// ---- 20_Product/10_BCF/10_Base/11_Com/01_Stringhandling/F_StringToTimeDate.TcPOU
// HI = parsing string 'Y-M-D, h:m:s.ms' or 'Y-M-D Th:m:s.ms' to TIMESTRUCT successful
FUNCTION PUBLIC F_StringToTimeDate : BOOL
(**************************************************************************************
 * 	Application		:	BoxControl Framework
 *	Revision		  :	$Revision: 461868 $
 *	Revision date	:	$Date: 1979-01-09 14:35:13 +0200 (Di., 09 Jan 1979) $
 *	Last changed by	:	$Author: b7lipim $
 *	URL				:	$URL: http://almscdc.swisslog.com/repo/SWPD/Development/BoxControlFramework/20_Release/branches/R1.x/01_Software/BCF/BCF/JumpStart/20_Product/10_BCF/10_Base/11_Com/12_DebugMsg/00_GVLs/DebugTextBlocks.TcGVL $
 *
 * ------------------------------------------------------------------------------------
 *	Copyright Swisslog [IP AG], Switzerland. All rights reserved.
 * 
 * ------------------------------------------------------------------------------------
 *	
 * 	Revision History: 
 *
 *  VERSION DATE         INITIALS     DESCRIPTION
 *  0.0     DD.MM.YYYY   (name)       (explain customized modifications)
 *
 **************************************************************************************)

(********************************************************************************************************************************)
VAR_INPUT
  DestStart             : POINTER TO BYTE                  := 0;     // = ADR(MyString)                    -> start position to concat
  DestEnd               : POINTER TO BYTE                  := 0;     // = ADR(MyString) + SIZEOF(MyString) -> buffer/string end
  (*----------------------------------------------------------------------------------------------------------------------------*)
  AllowInvalidChars     : BOOL                             := FALSE; // HI = ignore invalid char
END_VAR

(********************************************************************************************************************************)
VAR_OUTPUT
  Result                : TIMESTRUCT;                                     // parsing result
END_VAR

(********************************************************************************************************************************)
VAR
  Char                  : BYTE                             := 0;
  ItemType              : BYTE                             := UNDEF;
END_VAR

(********************************************************************************************************************************)
VAR CONSTANT
  UNDEF                 : BYTE := 0;
  YEAR                  : BYTE := 1;
  MONTH                 : BYTE := 2;
  DAY                   : BYTE := 3;
  HOUR                  : BYTE := 4;
  MINUTE                : BYTE := 5;
  SECOND                : BYTE := 6;
  MSEC                  : BYTE := 7;
END_VAR


(********************************************************************************************************************************)
(** check inputs ****************************************************************************************************************)
IF (    ( DestStart = 0 )
     OR ( DestEnd   = 0 )  )
THEN
  F_StringToTimeDate:= FALSE;
  RETURN;
END_IF




(********************************************************************************************************************************)
(********************************************************************************************************************************)
ItemType    := YEAR;

WHILE(DestStart^ <> 16#00)
DO
  Char     := DestStart^;
  DestStart:= DestStart + SIZEOF(DestStart^);
  (*-- numbers ----------------------------------------------------------------------------------------------*)
  IF (     ( Char >= 16#30 )
       AND ( Char <= 16#39 )  )
  THEN
    IF   (ItemType          = YEAR  ) THEN  Result.wYear        := (Result.wYear         * WORD#10) + BYTE_TO_WORD(Char - 16#30); 
    ELSIF(ItemType          = MONTH ) THEN  Result.wMonth       := (Result.wMonth        * WORD#10) + BYTE_TO_WORD(Char - 16#30);
    ELSIF(ItemType          = DAY   ) THEN  Result.wDay         := (Result.wDay          * WORD#10) + BYTE_TO_WORD(Char - 16#30);
    ELSIF(ItemType          = HOUR  ) THEN  Result.wHour        := (Result.wHour         * WORD#10) + BYTE_TO_WORD(Char - 16#30);
    ELSIF(ItemType          = MINUTE) THEN  Result.wMinute      := (Result.wMinute       * WORD#10) + BYTE_TO_WORD(Char - 16#30);
    ELSIF(ItemType          = SECOND) THEN  Result.wSecond      := (Result.wSecond       * WORD#10) + BYTE_TO_WORD(Char - 16#30);
    ELSIF(ItemType          = MSEC  ) THEN  Result.wMilliseconds:= (Result.wMilliseconds * WORD#10) + BYTE_TO_WORD(Char - 16#30);
    ELSIF(AllowInvalidChars = FALSE ) THEN  F_StringToTimeDate:= FALSE;  RETURN;
    END_IF

  (*-- separation during date -------------------------------------------------------------------------------*)
  ELSIF( Char = 16#2D ) (* '-' *)
  THEN
    IF   (ItemType          = YEAR  ) THEN  ItemType:= MONTH; 
    ELSIF(ItemType          = MONTH ) THEN  ItemType:= DAY;
    ELSIF(AllowInvalidChars = FALSE ) THEN  F_StringToTimeDate:= FALSE;  RETURN;
    END_IF

  (*-- separation date->time --------------------------------------------------------------------------------*)
  ELSIF(    ( Char = 16#2C )    (* ',' *)
         OR ( Char = 16#54 )  ) (* 'T' *)
  THEN
    IF   (ItemType          = DAY   ) THEN  ItemType:= HOUR; 
    ELSIF(AllowInvalidChars = FALSE ) THEN  F_StringToTimeDate:= FALSE;  RETURN;
    END_IF

  (*-- separation during time -------------------------------------------------------------------------------*)
  ELSIF( Char = 16#3A ) (* ':' *)
  THEN
    IF   (ItemType          = HOUR   ) THEN  ItemType:= MINUTE; 
    ELSIF(ItemType          = MINUTE ) THEN  ItemType:= SECOND;
    ELSIF(AllowInvalidChars = FALSE  ) THEN  F_StringToTimeDate:= FALSE;  RETURN;
    END_IF

  (*-- separation during time -------------------------------------------------------------------------------*)
  ELSIF( Char = 16#2E ) (* '.' *)
  THEN
    IF   (ItemType          = SECOND ) THEN  ItemType:= MSEC; 
    ELSIF(AllowInvalidChars = FALSE  ) THEN  F_StringToTimeDate:= FALSE;  RETURN;
    END_IF

  (*-- always ignore spaces ---------------------------------------------------------------------------------*)
  ELSIF( Char = 16#20) (* ' ' *)
  THEN
    CONTINUE;

  (*---------------------------------------------------------------------------------------------------------*)
  ELSIF (AllowInvalidChars = FALSE )
  THEN
    F_StringToTimeDate:= FALSE;
    RETURN;
  END_IF

END_WHILE




(********************************************************************************************************************************)
(** done ************************************************************************************************************************)
F_StringToTimeDate:=TRUE;

END_FUNCTION

// ---- 20_Product/30_Toolbox/12_StringStream/F_AssembleByteStream.TcPOU
FUNCTION F_AssembleByteStream  : BOOL
(**************************************************************************************
 * 	Application		:	BoxControl Framework
 *	Revision		:	$Revision: 404529 $
 *	Revision date	:	$Date: 2018-04-23 08:21:38 +0200 (Mo., 23 Apr 2018) $
 *	Last changed by	:	$Author: b7bolm $
 *	URL				:	$URL: http://almscdc.swisslog.com/repo/SWPD/Development/BoxControlFramework/20_Release/trunk/01_Software/BCF/BCF/JumpStart/30_Toolbox/12_StringStream/F_AssembleByteStream.TcPOU $
 *
 *	Purpose			:	Adds a String to an Address at position WritePointer.
 *						WritePointer starts at 0. After execution WritePointer returns
 *						WritePointer + Length of added data. This could be used to 
 *						call this function again to add a new data string directly
 *						after the last one.
 *
 * ------------------------------------------------------------------------------------
 *	Copyright Swisslog [IP AG], Switzerland. All rights reserved.
 * 
 * ------------------------------------------------------------------------------------
 *	
 * 	Revision History: 
 *
 * 	VERSION			DATE			INITIALS			DESCRIPTION
 *	0.1				01.01.2001		swl					Example
 *
 **************************************************************************************)
VAR_INPUT
	pSrc				: PVOID; // Address of source structure
	SrcLen				: UDINT; // Maximum size of source structure
	pDest				: PVOID; // Address of destination structure
	DestLen				: UDINT; // Maximum size of destination structure
END_VAR
VAR_IN_OUT
	WritePointer		: UDINT; // Address where the string should be added starting by 0, Returns Address + Length of added data 
END_VAR


// Validate inputs
IF WritePointer >= 0 AND
   WritePointer < DestLen AND
   DestLen > 0 AND
   pDest > 0 AND
   SrcLen > 0 THEN
   
   // Check if there is enough space to copy
   IF SrcLen <= DestLen - WritePointer THEN
		// Copy input stream to position (WriterPointer) of an address
		F_BlockCopy(
			pSrc := pSrc,
			LenSrc := SrcLen,
			pDest := pDest + WritePointer,
			LenDest := DestLen - WritePointer);
	
		// Update WritePointer 
		WritePointer := WritePointer + SrcLen;
		// Operation successful
		F_AssembleByteStream := TRUE;
	ELSE
		// Operation failed
		F_AssembleByteStream := FALSE;
	END_IF
ELSE
	// Operation failed
	F_AssembleByteStream := FALSE;
END_IF

END_FUNCTION

// ---- 20_Product/10_BCF/11_Conv/10_Base/13_GroupManager/FB_GroupManager.TcPOU
FUNCTION_BLOCK FB_GroupManager
(**************************************************************************************
 * 	Application		:	BoxControl Framework
 *	Revision		:	$Revision: 404529 $
 *	Revision date	:	$Date: 2018-04-23 08:21:38 +0200 (Mo., 23 Apr 2018) $
 *	Last changed by	:	$Author: b7bolm $
 *	URL				:	$URL: http://almscdc.swisslog.com/repo/SWPD/Development/BoxControlFramework/20_Release/trunk/01_Software/BCF/BCF/JumpStart/20_Product/10_App/14_Groups/10_Lib/10_Conv/FB_GroupManager.TcPOU $
 *
 *	Purpose			:	Group Manager - Administrates group states.
 *
 * ------------------------------------------------------------------------------------
 *	Copyright Swisslog [IP AG], Switzerland. All rights reserved.
 * 
 * ------------------------------------------------------------------------------------
 *	
 * 	Revision History: 
 *
 * 	VERSION			DATE			INITIALS			DESCRIPTION
 *	0.1				01.01.2001		swl					Example
 *
 **************************************************************************************)
VAR_INPUT
	Config						: ST_CFG_GroupManager; // GroupManager configuration
END_VAR

VAR
	Init						: BOOL := FALSE; // Instance is initialized
	
	fbDebugMsg					: FB_DebugMsg; // Debug Msg Manager (STACK) 
	DebugMsg					: T_MAXSTRING; // Debug msg
	OperationStateEmpty			: ST_PositionState;
	ElementReferenceTable		: ARRAY [E_BEGIN_ELEMENT..E_END_ELEMENT] OF ST_GroupManagerGroupMember;	// Referencetable - For each element, list the groups it belongs to
	GroupReferenceTable			: ARRAY [G_BEGIN_GROUP..G_END_GROUP] OF ST_GroupManagerElementMember; // Referencetable -  For each group, list the elements which belong to it *)
END_VAR

(**************************************************************************************************************
   Group Manager - Body never called!
***************************************************************************************************************)
;

METHOD M_GetGroupCmd : ST_PositionState
(**************************************************************************************
 * 	Application		:	BoxControl Framework
 *	Revision		:	$Revision: 404529 $
 *	Revision date	:	$Date: 2018-04-23 08:21:38 +0200 (Mo., 23 Apr 2018) $
 *	Last changed by	:	$Author: b7bolm $
 *	URL				:	$URL: http://almscdc.swisslog.com/repo/SWPD/Development/BoxControlFramework/20_Release/trunk/01_Software/BCF/BCF/JumpStart/20_Product/10_App/14_Groups/10_Lib/10_Conv/FB_GroupManager.TcPOU $
 *
 *	Purpose			:	M_GetGroupCmd
 *						An element requests its group state with this method. The Group Manager
 *						checks all groups which are related to this element, prioritize
 *						all states and returns the valid state to the element.
 *
 *						Additionally for all group types 'SG' (SwitchingGroup) the related
 *						Mode will be verified.
 *
 * ------------------------------------------------------------------------------------
 *	Copyright Swisslog [IP AG], Switzerland. All rights reserved.
 * 
 * ------------------------------------------------------------------------------------
 *	
 * 	Revision History: 
 *
 * 	VERSION			DATE			INITIALS			DESCRIPTION
 *	0.1				01.01.2001		swl					Example
 *
 **************************************************************************************)
VAR_INPUT
	meElementNumber		: E_ElementNumber; // The number of the element
END_VAR

VAR
	meGroupState		: E_PositionState; // enum group state
	meGroupMode			: E_PositionMode; // group mode
	meGroupNumber		: E_GroupNumber; // Group number
	mGroupState			: ST_PositionState; // group state
	eGroup				: E_GroupNumber; // Group iterator
	mLastValuesValid	: BOOL; // Last states are valid
END_VAR
// Initialize default values
meGroupState:= E_PositionState.UNKNOWN;
meGroupMode := E_PositionMode.UNKNOWN_MODE;
M_GetGroupCmd.eMode := meGroupMode;
M_GetGroupCmd.eState := meGroupState;
mLastValuesValid := FALSE;

// If the element number is valid 
IF (meElementNumber > E_BEGIN_ELEMENT) AND (meElementNumber < E_END_ELEMENT) THEN

	// Go trough all groups 
	FOR eGroup := G_BEGIN_GROUP + 1 TO G_END_GROUP - 1 DO
		// Get current group number
		meGroupNumber := ElementReferenceTable[meElementNumber].eMemberGroup[eGroup];
		
		
		// When the calling element is part of that group
		IF meGroupNumber > E_GroupNumber.G_BEGIN_GROUP THEN
			
			// Make sure the group is initilized, otherwise the reported state is maybe not valid
			IF F_IsGroupInitialized(eGroup) THEN
				mGroupState := F_GetGroupOperationState(eGroupNumber := meGroupNumber);
			ELSE
				mGroupState := OperationStateEmpty;
			END_IF
			
			(*
			Search for the highest prioritized state
			1. Unknown
			2. Stopped
			3. Stopping
			4. Starting
			5. Started
			
			Remark: An element can be part of multiple groups!
			*)
			IF mGroupState.eState = E_PositionState.UNKNOWN OR
               (meGroupState = E_PositionState.UNKNOWN AND mLastValuesValid) THEN
				
				meGroupState := E_PositionState.UNKNOWN;
			
			ELSIF mGroupState.eState = E_PositionState.STOPPED OR
                  (meGroupState = E_PositionState.STOPPED AND mLastValuesValid) THEN
			
				meGroupState := E_PositionState.STOPPED;
				
			ELSIF mGroupState.eState = E_PositionState.STOPPING OR
                  (meGroupState = E_PositionState.STOPPING AND mLastValuesValid) THEN
			
				meGroupState := E_PositionState.STOPPING;
				
			ELSIF mGroupState.eState = E_PositionState.STARTING OR
                  (meGroupState = E_PositionState.STARTING AND mLastValuesValid) THEN
			
				meGroupState := E_PositionState.STARTING;
				
			ELSIF mGroupState.eState = E_PositionState.STARTED OR
                  (meGroupState = E_PositionState.STARTED AND mLastValuesValid) THEN
			
				meGroupState := E_PositionState.STARTED;
			ELSE
				meGroupState := E_PositionState.UNKNOWN;
			END_IF
			
			
			(*
			Search for the highest prioritized mode
			1. Unknown
			2. OFF
			3. MANUAL
			4. SEMI_Auto
			5. Auto
			
			Remark: An element can be part of multiple groups!
			*)
			IF (meGroupMode = E_PositionMode.UNKNOWN_MODE AND mLastValuesValid) OR
			   mGroupState.eMode = E_PositionMode.UNKNOWN_MODE THEN

				meGroupMode := E_PositionMode.UNKNOWN_MODE;
				
			ELSIF (meGroupMode = E_PositionMode.OFF_MODE AND mLastValuesValid)OR
				  mGroupState.eMode = E_PositionMode.OFF_MODE THEN
			   
				meGroupMode := E_PositionMode.OFF_MODE;
					
			ELSIF (meGroupMode = E_PositionMode.MANUAL_MODE AND mLastValuesValid) OR
				  mGroupState.eMode = E_PositionMode.MANUAL_MODE THEN
			   
				meGroupMode := E_PositionMode.MANUAL_MODE;
				
			ELSIF (meGroupMode = E_PositionMode.SEMI_AUTO AND mLastValuesValid) OR
				  mGroupState.eMode = E_PositionMode.SEMI_AUTO THEN
			   
				meGroupMode := E_PositionMode.SEMI_AUTO;

			ELSIF (meGroupMode = E_PositionMode.AUTO_MODE AND mLastValuesValid) OR
				  mGroupState.eMode = E_PositionMode.AUTO_MODE THEN
				  
				meGroupMode := E_PositionMode.AUTO_MODE;
					
			// Otherwise the group has an invalid mode
			ELSE
				meGroupMode := E_PositionMode.UNKNOWN_MODE;
			END_IF
			
			// States of last group are valid
			mLastValuesValid := TRUE;
		END_IF
	END_FOR
	
	//Update output
	M_GetGroupCmd.eMode 		:= meGroupMode;
	M_GetGroupCmd.eState		:= meGroupState;
	M_GetGroupCmd.Info			:= mGroupState.Info;
	M_GetGroupCmd.InitRelease	:= mGroupState.InitRelease;
END_IF
END_METHOD

METHOD M_GetGroupMemberState : E_PositionState
(**************************************************************************************
 * 	Application		:	BoxControl Framework
 *	Revision		:	$Revision: 404529 $
 *	Revision date	:	$Date: 2018-04-23 08:21:38 +0200 (Mo., 23 Apr 2018) $
 *	Last changed by	:	$Author: b7bolm $
 *	URL				:	$URL: http://almscdc.swisslog.com/repo/SWPD/Development/BoxControlFramework/20_Release/trunk/01_Software/BCF/BCF/JumpStart/20_Product/10_App/14_Groups/10_Lib/10_Conv/FB_GroupManager.TcPOU $
 *
 *	Purpose			:	M_GetGroupMemberState
 *						A group requests the state of all appropriate elements. The
 *						Group Manager check all related elements and returns the summary
 *						of the states. If not all elements have the same state, an 
 *						"No state available" message will be returned.
 *
 * ------------------------------------------------------------------------------------
 *	Copyright Swisslog [IP AG], Switzerland. All rights reserved.
 * 
 * ------------------------------------------------------------------------------------
 *	
 * 	Revision History: 
 *
 * 	VERSION			DATE			INITIALS			DESCRIPTION
 *	0.1				01.01.2001		swl					Example
 *
 **************************************************************************************)
VAR_INPUT
	meGroupNumber 			: E_GroupNumber; // Requesting group number
END_VAR

VAR
	meElement				: E_ElementNumber; // Element iterator
	meLastGroupState		: E_PositionState; // Last group state, used for comparison
	meElementNumber			: E_ElementNumber; // Store ongoing element localy
	mFirstStateSaved		: BOOL; // Flag for storing first element state
	mElementState			: ST_PositionState; // Ongoing element state
END_VAR
// Initialize
M_GetGroupMemberState := E_PositionState.UNKNOWN;
meLastGroupState := E_PositionState.UNKNOWN;
mFirstStateSaved := FALSE;

// If the group number is valid
IF (meGroupNumber > G_BEGIN_GROUP) AND (meGroupNumber < G_END_GROUP) THEN

	// Go trough all elements	
	FOR meElement := E_BEGIN_ELEMENT + 1 TO E_END_ELEMENT - 1 DO
		// Store current element number
		meElementNumber := GroupReferenceTable[meGroupNumber].eMemberElement[meElement];
	
		// Only process records which have a valid element ID 
		IF meElementNumber <> E_BEGIN_ELEMENT THEN
				// Store internal data locally
				mElementState := F_GetElementOperationState(eElementNumber := meElementNumber);
			
				// If its not the first element
				IF mFirstStateSaved THEN
					// compare
					IF mElementState.eState <> meLastGroupState THEN
						// Return no unique state was found
						M_GetGroupMemberState := E_PositionState.UNKNOWN;
						RETURN;
					END_IF
				ELSE
					//Store 
					meLastGroupState := mElementState.eState;
					mFirstStateSaved := TRUE;
				END_IF
			END_IF
	END_FOR
	
	// If all members have the same state, return it
	M_GetGroupMemberState := meLastGroupState;
END_IF
END_METHOD

METHOD M_GroupMemberErrorPending : BOOL
(**************************************************************************************
 * 	Application		:	BoxControl Framework
 *	Revision		:	$Revision: 404529 $
 *	Revision date	:	$Date: 2018-04-23 08:21:38 +0200 (Mo., 23 Apr 2018) $
 *	Last changed by	:	$Author: b7bolm $
 *	URL				:	$URL: http://almscdc.swisslog.com/repo/SWPD/Development/BoxControlFramework/20_Release/trunk/01_Software/BCF/BCF/JumpStart/20_Product/10_App/14_Groups/10_Lib/10_Conv/FB_GroupManager.TcPOU $
 *
 *	Purpose			:	M_GroupMemberErrorPending
 *						A group requests the error state of all appropriate elements. 
 *						If one member is found with an error - True is returned.
 *
 * ------------------------------------------------------------------------------------
 *	Copyright Swisslog [IP AG], Switzerland. All rights reserved.
 * 
 * ------------------------------------------------------------------------------------
 *	
 * 	Revision History: 
 *
 * 	VERSION			DATE			INITIALS			DESCRIPTION
 *	0.1				01.01.2001		swl					Example
 *
 **************************************************************************************)
VAR_INPUT
	meGroupNumber 			: E_GroupNumber; // Requesting group number
END_VAR

VAR
	meElement				: E_ElementNumber; // Element iterator
	meElementNumber			: E_ElementNumber; // Store ongoing element localy
	mElementErrorData		: ST_ElementErrorStruct; // Ongoing element data
END_VAR

// Initialize
M_GroupMemberErrorPending := FALSE;

// If the group number is valid
IF (meGroupNumber > G_BEGIN_GROUP) AND (meGroupNumber < G_END_GROUP) THEN

	// Go trough all elements	
	FOR meElement := E_BEGIN_ELEMENT + 1 TO E_END_ELEMENT - 1 DO
		// Store current element number
		meElementNumber := GroupReferenceTable[meGroupNumber].eMemberElement[meElement];
	
		// Only process records which have a valid element ID 
		IF meElementNumber > E_ElementNumber.E_BEGIN_ELEMENT AND
           meElementNumber <  E_ElementNumber.E_END_ELEMENT THEN
			// Store internal data locally
			mElementErrorData := F_GetElementErrorData(eElementNumber := meElementNumber);
		
			// Check if the element or one of its functions is in error state
			IF mElementErrorData.Error.ErrorType = E_ErrorType.ERROR OR
			   mElementErrorData.FunctionErrorPending THEN
			   
				// Return 
				M_GroupMemberErrorPending := TRUE;
				EXIT;
			END_IF
		END_IF
	END_FOR
END_IF
END_METHOD

METHOD M_Init : BOOL
(**************************************************************************************
 * 	Application		:	BoxControl Framework
 *	Revision		:	$Revision: 404529 $
 *	Revision date	:	$Date: 2018-04-23 08:21:38 +0200 (Mo., 23 Apr 2018) $
 *	Last changed by	:	$Author: b7bolm $
 *	URL				:	$URL: http://almscdc.swisslog.com/repo/SWPD/Development/BoxControlFramework/20_Release/trunk/01_Software/BCF/BCF/JumpStart/20_Product/10_App/14_Groups/10_Lib/10_Conv/FB_GroupManager.TcPOU $
 *
 *	Purpose			:	M_Init
 *						Initialize GroupManager. 
 *
 * ------------------------------------------------------------------------------------
 *	Copyright Swisslog [IP AG], Switzerland. All rights reserved.
 * 
 * ------------------------------------------------------------------------------------
 *	
 * 	Revision History: 
 *
 * 	VERSION			DATE			INITIALS			DESCRIPTION
 *	0.1				01.01.2001		swl					Example
 *
 **************************************************************************************)
VAR_INPUT
	mInit				: BOOL; // True = Do init always , False = only if needed 
END_VAR

VAR
	eGroup				: E_GroupNumber; // Group iterator
	eElement			: E_ElementNumber; // Element iterator
	eGroupElement		: E_ElementNumber; // Element in this group
END_VAR
// If instance is not initialized
// or it has to be reinitialized
IF NOT Init OR mInit THEN
	// Populate the GroupTable 
	// For every group, copy the member elements to the GroupTable 
	FOR eGroup := G_BEGIN_GROUP TO G_END_GROUP DO
		FOR eElement := E_BEGIN_ELEMENT TO E_END_ELEMENT DO
			// Update GroupReferenceTable based on group manager configuration
			GroupReferenceTable[eGroup].eMemberElement[eElement] := Config.Group[eGroup].eMemberElement[eElement];
			
			IF Config.Group[eGroup].eMemberElement[eElement] > E_ElementNumber.E_BEGIN_ELEMENT THEN
				ElementReferenceTable[Config.Group[eGroup].eMemberElement[eElement]].eMemberGroup[eGroup] := eGroup;
			ELSE
				ElementReferenceTable[Config.Group[eGroup].eMemberElement[eElement]].eMemberGroup[eGroup] := E_GroupNumber.G_BEGIN_GROUP;
			END_IF
		END_FOR
	END_FOR

	// Initialization done
	Init := TRUE;
	
	// Return 
	M_Init := Init;
END_IF
END_METHOD

METHOD M_ResetMemberElements : BOOL
(**************************************************************************************
 * 	Application		:	BoxControl Framework
 *	Revision		:	$Revision: 404529 $
 *	Revision date	:	$Date: 2018-04-23 08:21:38 +0200 (Mo., 23 Apr 2018) $
 *	Last changed by	:	$Author: b7bolm $
 *	URL				:	$URL: http://almscdc.swisslog.com/repo/SWPD/Development/BoxControlFramework/20_Release/trunk/01_Software/BCF/BCF/JumpStart/20_Product/10_App/14_Groups/10_Lib/10_Conv/FB_GroupManager.TcPOU $
 *
 *	Purpose			:	M_ResetMemberElements - Send a reset command to all 
 *						appropriate elements of a group
 *
 * ------------------------------------------------------------------------------------
 *	Copyright Swisslog [IP AG], Switzerland. All rights reserved.
 * 
 * ------------------------------------------------------------------------------------
 *	
 * 	Revision History: 
 *
 * 	VERSION			DATE			INITIALS			DESCRIPTION
 *	0.1				01.01.2001		swl					Example
 *
 **************************************************************************************)
VAR_INPUT
	meGroupNumber 			: E_GroupNumber; // Requesting group number
END_VAR

VAR
	meElement				: E_ElementNumber; // Element iterator
	meElementNumber			: E_ElementNumber; // Store ongoing element localy
	mElementErrorData		: ST_ElementErrorStruct; // Ongoing element data
END_VAR

// Initialize
M_ResetMemberElements := FALSE;

// If the group number is valid
IF (meGroupNumber > G_BEGIN_GROUP) AND (meGroupNumber < G_END_GROUP) THEN

	// Go trough all elements	
	FOR meElement := E_BEGIN_ELEMENT + 1 TO E_END_ELEMENT - 1 DO
		// Store current element number
		meElementNumber := GroupReferenceTable[meGroupNumber].eMemberElement[meElement];
		
		// Only process records which have a valid element ID 
		IF meElementNumber > E_ElementNumber.E_BEGIN_ELEMENT AND
           meElementNumber <  E_ElementNumber.E_END_ELEMENT THEN
			// Store internal data locally
			mElementErrorData := F_GetElementErrorData(eElementNumber := meElementNumber);
		
			// Check if the element or one of its functions is in error state
			IF mElementErrorData.Error.ErrorType = E_ErrorType.ERROR OR
			   mElementErrorData.FunctionErrorPending THEN
				// Send reset command
				F_ResetElementError(
					eElementNumber := meElementNumber,
					ResetMembers := TRUE);
			END_IF
		END_IF
	END_FOR
END_IF
END_METHOD

END_FUNCTION_BLOCK

// ---- 20_Product/10_BCF/11_Conv/14_Groups/10_Helper/F_GetGroupOperationState.TcPOU
FUNCTION F_GetGroupOperationState : ST_PositionState
(**************************************************************************************
 * 	Application		:	BoxControl Framework
 *	Revision		:	$Revision: 404529 $
 *	Revision date	:	$Date: 2018-04-23 08:21:38 +0200 (Mo., 23 Apr 2018) $
 *	Last changed by	:	$Author: b7bolm $
 *	URL				:	$URL: http://almscdc.swisslog.com/repo/SWPD/Development/BoxControlFramework/20_Release/trunk/01_Software/BCF/BCF/JumpStart/20_Product/10_App/14_Groups/10_Lib/10_Conv/10_Functions/F_GetGroupOperationState.TcPOU $
 *
 *	Purpose			:	Returns group states
 *
 * ------------------------------------------------------------------------------------
 *	Copyright Swisslog [IP AG], Switzerland. All rights reserved.
 * 
 * ------------------------------------------------------------------------------------
 *	
 * 	Revision History: 
 *
 * 	VERSION			DATE			INITIALS			DESCRIPTION
 *	0.1				01.01.2001		swl					Example
 *
 **************************************************************************************)
VAR_INPUT
	eGroupNumber		: E_GroupNumber; // Group number
END_VAR



// Check if group number is valid
IF eGroupNumber > E_GroupNumber.G_BEGIN_GROUP AND
   eGroupNumber < E_GroupNumber.G_END_GROUP THEN

	// Check reference is valid
	IF __ISVALIDREF(GroupRegistry[eGroupNumber].rGroupData) THEN
   		// Return group state
   		F_GetGroupOperationState :=GroupRegistry[eGroupNumber].rGroupData.OperationState;
	END_IF
END_IF

END_FUNCTION

// ---- 20_Product/10_BCF/11_Conv/13_Elements/10_Helper/F_GetElementOperationState.TcPOU
FUNCTION F_GetElementOperationState : ST_PositionState
(**************************************************************************************
 * 	Application		:	BoxControl Framework
 *	Revision		:	$Revision: 404529 $
 *	Revision date	:	$Date: 2018-04-23 08:21:38 +0200 (Mo., 23 Apr 2018) $
 *	Last changed by	:	$Author: b7bolm $
 *	URL				:	$URL: http://almscdc.swisslog.com/repo/SWPD/Development/BoxControlFramework/20_Release/trunk/01_Software/BCF/BCF/JumpStart/20_Product/10_App/13_Elements/10_Lib/10_Conv/10_Functions/F_GetElementOperationState.TcPOU $
 *
 *	Purpose			:	Returns element states
 *
 * ------------------------------------------------------------------------------------
 *	Copyright Swisslog [IP AG], Switzerland. All rights reserved.
 * 
 * ------------------------------------------------------------------------------------
 *	
 * 	Revision History: 
 *
 * 	VERSION			DATE			INITIALS			DESCRIPTION
 *	0.1				01.01.2001		swl					Example
 *
 **************************************************************************************)
VAR_INPUT
	eElementNumber		: E_ElementNumber; // Element number
END_VAR



// Check if element number is valid
IF eElementNumber > E_ElementNumber.E_BEGIN_ELEMENT AND
   eElementNumber < E_ElementNumber.E_END_ELEMENT THEN
  
	// Check reference is valid
	IF __ISVALIDREF(ElementRegistry[eElementNumber].rElementData) THEN
   		// Return element state
   		F_GetElementOperationState :=ElementRegistry[eElementNumber].rElementData.OperationState;
	END_IF
END_IF

END_FUNCTION

// ---- 20_Product/10_BCF/11_Conv/13_Elements/10_Helper/F_GetElementErrorData.TcPOU
FUNCTION F_GetElementErrorData : ST_ElementErrorStruct
(**************************************************************************************
 * 	Application		:	BoxControl Framework
 *	Revision		:	$Revision: 404529 $
 *	Revision date	:	$Date: 2018-04-23 08:21:38 +0200 (Mo., 23 Apr 2018) $
 *	Last changed by	:	$Author: b7bolm $
 *	URL				:	$URL: http://almscdc.swisslog.com/repo/SWPD/Development/BoxControlFramework/20_Release/trunk/01_Software/BCF/BCF/JumpStart/20_Product/10_App/13_Elements/10_Lib/10_Conv/10_Functions/F_GetElementErrorData.TcPOU $
 *
 *	Purpose			:	Return element error data
 *
 * ------------------------------------------------------------------------------------
 *	Copyright Swisslog [IP AG], Switzerland. All rights reserved.
 * 
 * ------------------------------------------------------------------------------------
 *	
 * 	Revision History: 
 *
 * 	VERSION			DATE			INITIALS			DESCRIPTION
 *	0.1				01.01.2001		swl					Example
 *
 **************************************************************************************)
VAR_INPUT
	eElementNumber		: E_ElementNumber; // Element number
END_VAR


// Check if element number is valid
IF eElementNumber > E_ElementNumber.E_BEGIN_ELEMENT AND
   eElementNumber < E_ElementNumber.E_END_ELEMENT THEN
  
	// Check reference is valid
	IF __ISVALIDREF(ElementRegistry[eElementNumber].rElementData) THEN
   		// Return error data
   		F_GetElementErrorData := ElementRegistry[eElementNumber].rElementData.ErrorData;
	END_IF
END_IF

END_FUNCTION

// ---- 20_Product/10_BCF/11_Conv/13_Elements/10_Helper/F_ResetElementError.TcPOU
FUNCTION F_ResetElementError : BOOL
(**************************************************************************************
 * 	Application		:	BoxControl Framework
 *	Revision		:	$Revision: 404529 $
 *	Revision date	:	$Date: 2018-04-23 08:21:38 +0200 (Mo., 23 Apr 2018) $
 *	Last changed by	:	$Author: b7bolm $
 *	URL				:	$URL: http://almscdc.swisslog.com/repo/SWPD/Development/BoxControlFramework/20_Release/trunk/01_Software/BCF/BCF/JumpStart/20_Product/10_App/13_Elements/10_Lib/10_Conv/10_Functions/F_ResetElementError.TcPOU $
 *
 *	Purpose			:	Reset element error
 *
 * ------------------------------------------------------------------------------------
 *	Copyright Swisslog [IP AG], Switzerland. All rights reserved.
 * 
 * ------------------------------------------------------------------------------------
 *	
 * 	Revision History: 
 *
 * 	VERSION			DATE			INITIALS			DESCRIPTION
 *	0.1				01.01.2001		swl					Example
 *
 **************************************************************************************)
VAR_INPUT
	eElementNumber		: E_ElementNumber; // Element number to send reset
	ResetMembers		: BOOL; // Reset members as well
END_VAR


// Check if element number is valid
IF eElementNumber > E_ElementNumber.E_BEGIN_ELEMENT AND
   eElementNumber < E_ElementNumber.E_END_ELEMENT THEN

	// If reference is valid
	IF __ISVALIDREF(ElementRegistry[eElementNumber].rElement) THEN
		// Reset function
		ElementRegistry[eElementNumber].rElement.M_ResetError(mResetMembers := ResetMembers);
	END_IF
END_IF

END_FUNCTION

// ---- 20_Product/10_BCF/11_Conv/11_Com/11_ITC/FB_ITC_Conveyor.TcPOU
FUNCTION_BLOCK FB_ITC_Conveyor IMPLEMENTS ITF_ITC
(**************************************************************************************
 *  Application     :   BoxControl Framework
 *  Revision date   :   $Date: 2021-04-08 12:45:11 +0200 (tor, 08 apr 2021) $
 *  Author          :   CDC
 *	Purpose			:	ITC - Message Manager.
 *						Represents the interface between the application and the 
 *						communication. Serves as abstract layer to ensure application
 *						independency.
 * ------------------------------------------------------------------------------------
 *  © Swisslog AG
 *  Swisslog is not liable for any usage of this source code that is not agreed 
 *  on between Swisslog and the other party. The mandatory legal liability remains 
 *  unaffected.
 * ------------------------------------------------------------------------------------
 *  Revision History: 
 *
 *  VERSION DATE         INITIALS     DESCRIPTION
 *  0.0     DD.MM.YYYY   (name)       (explain customized modifications)
 *
 **************************************************************************************)
VAR_INPUT
	Config			: ST_CFG_ITC_ManagerConv; // Config
END_VAR

VAR
	Init			: BOOL; // Initialized
	fbDebugMsg		: FB_DebugMsg; // Debug instance
	DebugMsg		: T_MAXSTRING; // Debug msg
	Idx				: INT; // Index for general usage 
	eMsgType		: E_ITC_MsgTypeConv; // Message type conveyor
	Position		: ST_PositionIdent;
	SDI				: ST_ITC_SDI; // SDI
	GVR				: ST_ITC_GVR; // GVR
	ISR				: ST_ITC_ISR; // ISR
	TTC				: ST_ITC_TTC; // TTC
	TDR				: ST_ITC_TDR; // TDR
	FCQ				: ST_ITC_FCQ; // FCQ
	FSR				: ST_ITC_FSR; // FSR
	FSR_Empty		: ST_ITC_FSR; // FSR empty
	SCR				: ST_ITC_SCR; // SCR
	SSR				: ST_ITC_SSR; // SSR
	SSR_Empty		: ST_ITC_SSR; // SSR empty
	GCR				: ST_ITC_GCR; // GCR
	GSR				: ST_ITC_GSR; // GSR
	GSR_Empty		: ST_ITC_GSR; // GSR empty
	ECR				: ST_ITC_ECR; // ECR
	ESR				: ST_ITC_ESR; // ESR
	ESR_Empty		: ST_ITC_ESR; // ESR empty
	FCR				: ST_ITC_FCR; // FCR
	MCR				: ST_ITC_MCR; // MCR
	MCR_Empty		: ST_ITC_MCR; // MCR empty
	SIR				: ST_ITC_SIR; // SIR
	TUR				: ST_ITC_TUR; // TUR
	GDR				: ST_ITC_GDR; // GDR
	GDR_Empty		: ST_ITC_GDR; // GDR empty
	DAR				: ST_ITC_DAR; // DAR
	DAR_Empty		: ST_ITC_DAR; // DAR empty
	Data			: ST_ITC_GeneralData; // General data
	RAC				: ST_ITC_RAC; // RAC
	RDR				: ST_ITC_RDR; // RDR
END_VAR

VAR PERSISTENT
	Settings			: ST_CFG_ITC_ManagerConv; // Active configuration
END_VAR

(**************************************************************************************************************
   Body never called!
***************************************************************************************************************)
;

{attribute 'object_name' := 'M_AddData'}
METHOD M_AddData : BOOL
(**************************************************************************************
 * 	Application		:	BoxControl Framework
 *	Revision		:	$Revision: 474929 $
 *	Revision date	:	$Date: 2021-04-08 12:45:11 +0200 (tor, 08 apr 2021) $
 *	Last changed by	:	$Author: b7gessa $
 *	URL				:	$URL: http://almscdc.swisslog.com/repo/SWPD/Development/BoxControlFramework/20_Release/tags/R1.12.0/01_Software/BCF/BCF/JumpStart/20_Product/10_BCF/11_Conv/11_Com/11_ITC/FB_ITC_Conveyor.TcPOU $
 *
 *	Purpose			:	Add data to the system
 *
 * ------------------------------------------------------------------------------------
 *	Copyright Swisslog [IP AG], Switzerland. All rights reserved.
 * 
 * ------------------------------------------------------------------------------------
 *	
 * 	Revision History: 
 *
 * 	VERSION			DATE			INITIALS			DESCRIPTION
 *	0.1				01.01.2001		swl					Example
 *
 **************************************************************************************)
VAR_INPUT
	meChannelSrc	: E_MFCS_Channel;
	mMsgType		: INT;
	mpData			: PVOID;
	mLen			: UDINT;
END_VAR

M_AddData := FALSE;
// Translate type to enumeration
eMsgType := mMsgType;

// Go to corresponding type
CASE eMsgType OF
	(****************************************************
	  No Message type
	*****************************************************)	
	E_ITC_MsgTypeConv.NO_MESSAGE_TYPE:
		;
	
	(****************************************************
	  Visualization information request
	*****************************************************)	
	E_ITC_MsgTypeConv.VISUALIZATION_INFORMATION_REQUEST:
		// Process
		M_AddData := M_ProcessVIQ(
						meChannelSrc := meChannelSrc,
						mpVIQ := mpData,
						mLen := mLen);
		
	(****************************************************
	  Digital input request
	*****************************************************)	
	E_ITC_MsgTypeConv.DIGITAL_INPUT_REQUEST:
		// Process
		M_AddData := M_ProcessDIQ(
						meChannelSrc := meChannelSrc);
		
	(****************************************************
	  Element control request
	*****************************************************)
	E_ITC_MsgTypeConv.ELEMENT_CONTROL_REQUEST:
		// Process
		M_AddData := M_ProcessECQ(
						meChannelSrc := meChannelSrc,
						mpECQ		 := mpData,
						mLen 		 := mLen);
	
	(****************************************************
	  Element status request
	*****************************************************)		
	E_ITC_MsgTypeConv.ELEMENT_STATUS_REQUEST:
		// Process
		M_AddData := M_ProcessESQ(
						meChannelSrc := meChannelSrc,
						mpESQ		 := mpData,
						mLen 	     := mLen);
		
	(****************************************************
	  Function control request
	*****************************************************)	
	E_ITC_MsgTypeConv.FUNCTION_CONTROL_REQUEST:
		// Process
		M_AddData := M_ProcessFCQ(
						meChannelSrc := meChannelSrc,
						mpFCQ		 := mpData,
						mLen 		 := mLen);
		
	(****************************************************
	  Function status request
	*****************************************************)	
	E_ITC_MsgTypeConv.FUNCTION_STATUS_REQUEST:
		// Process
		M_AddData := M_ProcessFSQ(
						meChannelSrc := meChannelSrc,
						mpFSQ		 := mpData,
						mLen 		 := mLen);
						
	(****************************************************
	  Group control request
	*****************************************************)				
	E_ITC_MsgTypeConv.GROUP_CONTROL_REQUEST:
		// Process
		M_AddData := M_ProcessGCQ(
						meChannelSrc := meChannelSrc,
						mpGCQ		 := mpData,
						mLen 		 := mLen);

	(****************************************************
	  Group status request
	*****************************************************)	
	E_ITC_MsgTypeConv.GROUP_STATUS_REQUEST:
		// Process
		M_AddData := M_ProcessGSQ(
						meChannelSrc := meChannelSrc,
						mpGSQ		 := mpData,
						mLen 		 := mLen);
		
	(****************************************************
	  Global variable request
	*****************************************************)	
	E_ITC_MsgTypeConv.GLOBAL_VARIABLE_REQUEST:
		// Process
		M_AddData := M_ProcessGVQ(
						meChannelSrc := meChannelSrc,
						mpGVQ := mpData,
						mLen := mLen);
						
	(****************************************************
	  IRQ request
	*****************************************************)	
	E_ITC_MsgTypeConv.I_O_STATUS_REQUEST:
		// Process
		M_AddData := M_ProcessIRQ(
						meChannelSrc := meChannelSrc,
						mpIRQ		 := mpData,
						mLen 	     := mLen);
		
	(****************************************************
	  Manual control request
	*****************************************************)					
	E_ITC_MsgTypeConv.MANUAL_CONTROL_REQUEST:
		// Process
		M_AddData := M_ProcessMCQ(
						meChannelSrc := meChannelSrc,
						mpMCQ		 := mpData,
						mLen 		 := mLen);
		
	(****************************************************
	  Robot action assignement
	*****************************************************)					
	E_ITC_MsgTypeConv.ROBOT_ACTION_ASSIGNMENT:
		// Process
		M_AddData := M_ProcessRAA(
						meChannelSrc := meChannelSrc,
						mpRAA		 := mpData,
						mLen 		 := mLen);		
				
	(****************************************************
	  Robot delete request
	*****************************************************)					
	E_ITC_MsgTypeConv.ROBOT_DELETE_REQUEST:
		// Process
		M_AddData := M_ProcessRDQ(
						meChannelSrc := meChannelSrc,
						mpRDQ		 := mpData,
						mLen 		 := mLen);	
			
	(****************************************************
	  Subsystem control request
	*****************************************************)				
	E_ITC_MsgTypeConv.SUBSYSTEM_CONTROL_REQUEST:
		// Process
		M_AddData := M_ProcessSCQ(
						meChannelSrc := meChannelSrc,
						mpSCQ		 := mpData,
						mLen 		 := mLen);
		
	(****************************************************
	  Set digital output
	*****************************************************)				
	E_ITC_MsgTypeConv.SET_DIGITAL_OUTPUT:
		// Process
		M_AddData := M_ProcessSDO(
						meChannelSrc := meChannelSrc,
						mpSDO		 := mpData,
						mLen 		 := mLen);
		
	(****************************************************
	  Scanner information request
	*****************************************************)				
	E_ITC_MsgTypeConv.SCANNER_INFORMATION_REQUEST:
		// Process
		M_AddData := M_ProcessSIQ(
						meChannelSrc := meChannelSrc,
						mpSIQ		 := mpData,
						mLen 		 := mLen);
		
	(****************************************************
	  Subsystem status request
	*****************************************************)			
	E_ITC_MsgTypeConv.SUBSYSTEM_STATUS_REQUEST:
		// Process
		M_AddData := M_ProcessSSQ(
						meChannelSrc := meChannelSrc,
						mpSSQ		 := mpData,
						mLen 		 := mLen);
		
	(****************************************************
	  Task delete request
	*****************************************************)			
	E_ITC_MsgTypeConv.TASK_DELETE_REQUEST:
		// Process
		M_AddData := M_ProcessTDQ(
						meChannelSrc := meChannelSrc,
						mpTDQ		 := mpData,
						mLen 		 := mLen);
		
	(****************************************************
	  Transport task assignment
	*****************************************************)	
	E_ITC_MsgTypeConv.TRANSPORT_TASK_ASSIGNMENT:
		// Process
		M_AddData := M_ProcessTTA(
						meChannelSrc := meChannelSrc,
						mpTTA		 := mpData,
						mLen 		 := mLen);
		
	(****************************************************
	  Transport unit request
	*****************************************************)	
	E_ITC_MsgTypeConv.TRANSPORT_UNIT_REQUEST:
		// Process
		M_AddData := M_ProcessTUQ(
						meChannelSrc := meChannelSrc,
						mpTUQ		 := mpData,
						mLen 	     := mLen);

	(****************************************************
	  Add TU data index into function
	*****************************************************)	
	E_ITC_MsgTypeConv.ADD_TU_DATA:
		// Process
		M_AddData := M_AddTUData(
						meChannelSrc := meChannelSrc,
						mpAddTU_Data		 := mpData);					


						
	(****************************************************
		Data Aquisition Request 
	*****************************************************)	
	E_ITC_MsgTypeConv.DATA_ACQUISITION_REQUEST:
		// Process
		M_AddData := M_ProcessDAQ(
						meChannelSrc := meChannelSrc,
						mpDAQ		 := mpData,
						mLen 	     := mLen);
	(****************************************************
		Gathered Data  Request 
	*****************************************************)	
	E_ITC_MsgTypeConv.GATHERED_DATA_REQUEST:
		// Process
		M_AddData := M_ProcessGDQ(
						meChannelSrc := meChannelSrc,
						mpGDQ		 := mpData,
						mLen 	     := mLen);				
ELSE
	// Unknown type
	DebugMsg := 'Unknown message type received';
	fbDebugMsg.M_SendErrorMsg(mMessage := DebugMsg);		
END_CASE
END_METHOD

METHOD PROTECTED M_AddTUData : BOOL

(**************************************************************************************
 * 	Application		:	BoxControl Framework
 *	Revision		:	$Revision: 474929 $
 *	Revision date	:	$Date: 2021-04-08 12:45:11 +0200 (tor, 08 apr 2021) $
 *	Last changed by	:	$Author: b7gessa $
 *	URL				:	$URL: http://almscdc.swisslog.com/repo/SWPD/Development/BoxControlFramework/20_Release/tags/R1.12.0/01_Software/BCF/BCF/JumpStart/20_Product/10_BCF/11_Conv/11_Com/11_ITC/FB_ITC_Conveyor.TcPOU $
 *
 *	Purpose			:	Process a received Digital Input Request telegram.
 *
 * ------------------------------------------------------------------------------------
 *	Copyright Swisslog [IP AG], Switzerland. All rights reserved.
 * 
 * ------------------------------------------------------------------------------------
 *	
 * 	Revision History: 
 *
 * 	VERSION			DATE			INITIALS			DESCRIPTION
 *	0.1				01.01.2001		swl					Example
 *
 **************************************************************************************)
VAR_INPUT
	meChannelSrc		: E_MFCS_Channel; // Source communicaton channel
	mpAddTU_Data		: POINTER TO ST_ITC_ADD_TU_DATA; // Pointer to SCQ
END_VAR
Data.Init := TRUE;
Data.TU_DataIndex := mpAddTU_Data^.TU_DataIndex;
Data.ZoneNumber := mpAddTU_Data^.ZoneNumber;
Data.Position := '';

// Forward to position
M_AddTUData := M_ProcessToFunction(
	meFunctionNumber	:= mpAddTU_Data^.eFunctionNumber, 
	meChannelSrc		:= meChannelSrc, 
	mMsgType			:= E_ITC_MsgTypeConv.ADD_TU_DATA,
	mpData				:= ADR(Data), 
	mLen				:= SIZEOF(Data));
END_METHOD

{attribute 'object_name' := 'M_CallITC_Service'}
METHOD M_CallITC_Service : BOOL
VAR
	mIdx : INT;
END_VAR
(**************************************************************************************************************
 	Initialization
***************************************************************************************************************)
M_Init(FALSE);

(**************************************************************************************************************
  Monitor SDI Signals
***************************************************************************************************************)
FOR mIdx := 1 TO Settings.SDI_Limit DO
	// SDI signal is enabled 
	IF SDISignalNumber[mIdx].Enabled THEN
		// SDI signal changed state 
		IF SDISignalNumber[mIdx].State <> SDISignalNumber[mIdx].LastState THEN
			// Send SDI
			F_ITC_SendSDI(
				eChannelSrc		:= 0, 
				SignalNumber	:= mIdx, 
				SignalState		:= SDISignalNumber[mIdx].State, 
				eReturnCode		:= E_ErrorConv.NO_ERROR_CODE);
				
			// Update state
			SDISignalNumber[mIdx].LastState := SDISignalNumber[mIdx].State;
		END_IF
	END_IF
END_FOR
END_METHOD

METHOD M_Init : BOOL
(**************************************************************************************
 * 	Application		:	BoxControl Framework
 *	Revision		:	$Revision: 474929 $
 *	Revision date	:	$Date: 2021-04-08 12:45:11 +0200 (tor, 08 apr 2021) $
 *	Last changed by	:	$Author: b7gessa $
 *	URL				:	$URL: http://almscdc.swisslog.com/repo/SWPD/Development/BoxControlFramework/20_Release/tags/R1.12.0/01_Software/BCF/BCF/JumpStart/20_Product/10_BCF/11_Conv/11_Com/11_ITC/FB_ITC_Conveyor.TcPOU $
 *
 *	Purpose			:	Initialize.
 *
 * ------------------------------------------------------------------------------------
 *	Copyright Swisslog [IP AG], Switzerland. All rights reserved.
 * 
 * ------------------------------------------------------------------------------------
 *	
 * 	Revision History: 
 *
 * 	VERSION			DATE			INITIALS			DESCRIPTION
 *	0.1				01.01.2001		swl					Example
 *
 **************************************************************************************)
VAR_INPUT
	mInit		: BOOL; // Force init
END_VAR
// If instance is not initialized or init is forced
IF mInit OR NOT Init THEN
	// Update configuration
	Settings := Config;
	
	// Send log message
    fbDebugMsg.M_SendInfoMsg('Initialization done');
		
	// Init done
    Init := TRUE;
END_IF
END_METHOD

METHOD PRIVATE M_ProcessDAQ : BOOL
(**************************************************************************************
 * 	Application		:	BoxControl Framework
 *	Revision		:	$Revision: 474929 $
 *	Revision date	:	$Date: 2021-04-08 12:45:11 +0200 (tor, 08 apr 2021) $
 *	Last changed by	:	$Author: b7gessa $
 *	URL				:	$URL: http://almscdc.swisslog.com/repo/SWPD/Development/BoxControlFramework/20_Release/tags/R1.12.0/01_Software/BCF/BCF/JumpStart/20_Product/10_BCF/11_Conv/11_Com/11_ITC/FB_ITC_Conveyor.TcPOU $
 *
 *	Purpose			:	Process a received Data Aquisition telegram.
 *
 * ------------------------------------------------------------------------------------
 *	Copyright Swisslog [IP AG], Switzerland. All rights reserved.
 * 
 * ------------------------------------------------------------------------------------
 *	
 * 	Revision History: 
 *
 * 	VERSION			DATE			INITIALS			DESCRIPTION
 *	0.1				01.01.2001		swl					Example
 *
 **************************************************************************************)
VAR_INPUT
	meChannelSrc		: E_MFCS_Channel; // Source communicaton channel
	mpDAQ				: POINTER TO ST_ITC_DAQ; // Pointer to DAQ
	mLen				: UDINT; // Data length
END_VAR
VAR
	meFunctionPosition		: ST_PositionIdent; // Position
	meGroupNumber			: E_GroupNumber; // Group
	meElementNumber			: E_ElementNumber;//Element Number
	meSubsystem				: BOOL;	//Subsystem
	mReturnCode				: E_ErrorConv; // Error code

END_VAR
// Initialize
M_ProcessDAQ:= TRUE;

//Check where position is
meFunctionPosition := F_SearchFunctionPosition(Position := mpDAQ^.Position);
meElementNumber    := F_SearchElementPosition(ElementName := mpDAQ^.Position);
meGroupNumber      := F_SearchGroupNumber(GroupName := mpDAQ^.Position);
meSubsystem 	   := F_EqualSisNames(Name1 := SubsystemRegistry.SubSystemName,
									Name2 := mpDAQ^.Position);

// Check if Function Number is valid
IF meFunctionPosition.eFunctionNumber >F_BEGIN_FUNCTION AND
	meFunctionPosition.eFunctionNumber <F_END_FUNCTION THEN 
    // Forward to Function
	M_ProcessDAQ := M_ProcessToFunction(
						meFunctionNumber:= 	meFunctionPosition.eFunctionNumber, // Position
						meChannelSrc	:= meChannelSrc, 
						mpData			:= mpDAQ, 
						mMsgType		:= E_ITC_MsgTypeConv.DATA_ACQUISITION_REQUEST,
						mLen			:= mLen);
// Check if DAQ was sent to an Element	
ELSIF meElementNumber > E_ElementNumber.E_BEGIN_ELEMENT AND 
      meElementNumber < E_ElementNumber.E_END_ELEMENT AND
      meFunctionPosition.eFunctionNumber = F_BEGIN_FUNCTION AND
      meFunctionPosition.ZoneNumber = 0 THEN 
		// Forward to element
		M_ProcessDAQ := M_ProcessToElement(
						meElementNumber	:= meElementNumber, 
						meChannelSrc	:= meChannelSrc, 
						mpData			:= mpDAQ, 
						mMsgType		:= E_ITC_MsgTypeConv.DATA_ACQUISITION_REQUEST,
						mLen			:= mLen);
// Check if DAQ was sent to a Group					
ELSIF  meGroupNumber > E_GroupNumber.G_BEGIN_GROUP AND 
   		meGroupNumber < E_GroupNumber.G_END_GROUP   AND
		meElementNumber 					= E_BEGIN_ELEMENT AND 
      	meFunctionPosition.eFunctionNumber 	= F_BEGIN_FUNCTION AND
      	meFunctionPosition.ZoneNumber 		= 0 THEN 	   
		// Forward to Group
		M_ProcessDAQ := M_ProcessToGroup(
							meGroupNumber	:= meGroupNumber, // Groupnumber
							meChannelSrc	:= meChannelSrc, 
							mpData			:= mpDAQ, 
							mMsgType		:= E_ITC_MsgTypeConv.DATA_ACQUISITION_REQUEST,
							mLen			:= mLen);
// Check if DAQ was sent to a SubSystem
ELSIF  meSubsystem AND
	   meGroupNumber = G_BEGIN_GROUP AND
	   meElementNumber = E_BEGIN_ELEMENT AND 
	   meFunctionPosition.eFunctionNumber = F_BEGIN_FUNCTION AND
	   meFunctionPosition.ZoneNumber = 0 THEN 	   		
	// Forward to Subsytem						
	M_ProcessDAQ := M_ProcessToSubsystem(
						meChannelSrc	:= meChannelSrc, 
						mpData			:= mpDAQ, 
						mMsgType		:= E_ITC_MsgTypeConv.DATA_ACQUISITION_REQUEST,
						mLen			:= mLen);					
ELSE
	//Unknown position send DAR with Error Report	
	DAR := DAR_Empty;
	// DAR
	DAR.Position	:= mpDAQ^.Position;
	DAR.eErrorCode	:= E_ErrorConv.ELEMENTNUMBER_UNKNOWN;

	// Reject telegram	
	M_SendData(
		meChannel := meChannelSrc,
		mMsgType  := E_ITC_MsgTypeConv.DATA_ACQUISITION_REPORT,
		mpData    := ADR(DAR),
		mLen	  := SIZEOF(DAR));
		
	// Unknown Position name received
	DebugMsg := CONCAT('DAQ - unknown Position name received: ', mpDAQ^.Position);
	fbDebugMsg.M_SendErrorMsg(mMessage := DebugMsg);
END_IF
END_METHOD

METHOD PROTECTED M_ProcessDIQ : BOOL
(**************************************************************************************
 * 	Application		:	BoxControl Framework
 *	Revision		:	$Revision: 474929 $
 *	Revision date	:	$Date: 2021-04-08 12:45:11 +0200 (tor, 08 apr 2021) $
 *	Last changed by	:	$Author: b7gessa $
 *	URL				:	$URL: http://almscdc.swisslog.com/repo/SWPD/Development/BoxControlFramework/20_Release/tags/R1.12.0/01_Software/BCF/BCF/JumpStart/20_Product/10_BCF/11_Conv/11_Com/11_ITC/FB_ITC_Conveyor.TcPOU $
 *
 *	Purpose			:	Process a received Digital Input Request telegram.
 *
 * ------------------------------------------------------------------------------------
 *	Copyright Swisslog [IP AG], Switzerland. All rights reserved.
 * 
 * ------------------------------------------------------------------------------------
 *	
 * 	Revision History: 
 *
 * 	VERSION			DATE			INITIALS			DESCRIPTION
 *	0.1				01.01.2001		swl					Example
 *
 **************************************************************************************)
VAR_INPUT
	meChannelSrc			: E_MFCS_Channel; // Source communicaton channel
END_VAR
// Compose an SDI telegram for every enabled SDI signal
FOR Idx := 1 TO NUMBER_OF_SDI_SIGNALS DO
	// For all enabled SDI SignalNumbers
	IF SDISignalNumber[Idx].Enabled THEN
		// Collect data
		SDI.SignalNumber := Idx;
		SDI.SignalState  := SDISignalNumber[Idx].State;
		SDI.ReturnCode	 := E_ErrorConv.NO_ERROR_CODE;
	
		M_SendData(
			meChannel := meChannelSrc, 
			mMsgType  := E_ITC_MsgTypeConv.SEND_DIGITAL_INPUT, 
			mpData    := ADR(SDI),
			mLen	  := SIZEOF(SDI));
	END_IF
END_FOR

// Telegram processed
M_ProcessDIQ := TRUE;
END_METHOD

METHOD PROTECTED M_ProcessECQ : BOOL
(**************************************************************************************
 * 	Application		:	BoxControl Framework
 *	Revision		:	$Revision: 474929 $
 *	Revision date	:	$Date: 2021-04-08 12:45:11 +0200 (tor, 08 apr 2021) $
 *	Last changed by	:	$Author: b7gessa $
 *	URL				:	$URL: http://almscdc.swisslog.com/repo/SWPD/Development/BoxControlFramework/20_Release/tags/R1.12.0/01_Software/BCF/BCF/JumpStart/20_Product/10_BCF/11_Conv/11_Com/11_ITC/FB_ITC_Conveyor.TcPOU $
 *
 *	Purpose			:	Process a received Element Control Request 
 *
 * ------------------------------------------------------------------------------------
 *	Copyright Swisslog [IP AG], Switzerland. All rights reserved.
 * 
 * ------------------------------------------------------------------------------------
 *	
 * 	Revision History: 
 *
 * 	VERSION			DATE			INITIALS			DESCRIPTION
 *	0.1				01.01.2001		swl					Example
 *
 **************************************************************************************)
VAR_INPUT
	meChannelSrc		: E_MFCS_Channel; // Source communicaton channel
	mpECQ				: POINTER TO ST_ITC_ECQ; // Pointer to ECQ
	mLen				: UDINT; // Data length
END_VAR

VAR
	meElementNumber		: E_ElementNumber; // Element number
END_VAR
// Initialize
M_ProcessECQ := TRUE;

// Try getting enum
meElementNumber := F_SearchElementPosition(ElementName := mpECQ^.Position);

// Check if ElementNumber is valid
IF meElementNumber > E_ElementNumber.E_BEGIN_ELEMENT AND 
   meElementNumber < E_ElementNumber.E_END_ELEMENT THEN
			
	// Forward to element
	M_ProcessECQ := M_ProcessToElement(
						meElementNumber	:= meElementNumber, 
						meChannelSrc	:= meChannelSrc, 
						mMsgType		:= E_ITC_MsgTypeConv.ELEMENT_CONTROL_REQUEST,
						mpData			:= mpECQ, 
						mLen			:= mLen);
						
ELSE
	// Unknown Position name received
	// ECR
	ECR.Position	:= mpECQ^.Position;
	ECR.Code		:= mpECQ^.Code;
	ECR.Variable	:= mpECQ^.Variable;
	ECR.ReturnCode	:= E_ErrorConv.ELEMENTNUMBER_UNKNOWN;

	// Reject telegram	
	M_SendData(
		meChannel := meChannelSrc,
		mMsgType  := E_ITC_MsgTypeConv.ELEMENT_CONTROL_REPLY,
		mpData    := ADR(ECR),
		mLen	  := SIZEOF(ECR));
		
	// Unknown Position name received
	DebugMsg := CONCAT('ECQ - unknown Position name received: ', mpECQ^.Position);
	fbDebugMsg.M_SendErrorMsg(mMessage := DebugMsg);
END_IF
END_METHOD

METHOD PROTECTED M_ProcessESQ : BOOL
(**************************************************************************************
 * 	Application		:	BoxControl Framework
 *	Revision		:	$Revision: 474929 $
 *	Revision date	:	$Date: 2021-04-08 12:45:11 +0200 (tor, 08 apr 2021) $
 *	Last changed by	:	$Author: b7gessa $
 *	URL				:	$URL: http://almscdc.swisslog.com/repo/SWPD/Development/BoxControlFramework/20_Release/tags/R1.12.0/01_Software/BCF/BCF/JumpStart/20_Product/10_BCF/11_Conv/11_Com/11_ITC/FB_ITC_Conveyor.TcPOU $
 *
 *	Purpose			:	Process a received Element Status Request telegram.
 *
 * ------------------------------------------------------------------------------------
 *	Copyright Swisslog [IP AG], Switzerland. All rights reserved.
 * 
 * ------------------------------------------------------------------------------------
 *	
 * 	Revision History: 
 *
 * 	VERSION			DATE			INITIALS			DESCRIPTION
 *	0.1				01.01.2001		swl					Example
 *
 **************************************************************************************)
VAR_INPUT
	meChannelSrc		: E_MFCS_Channel; // Source communicaton channel
	mpESQ				: POINTER TO ST_ITC_ESQ; // Pointer to ESQ
	mLen				: UDINT; // Data length
END_VAR

VAR
	meElementNumber		: E_ElementNumber; // Element number
END_VAR
// Initialize
M_ProcessESQ := TRUE;

// Try getting enum
meElementNumber := F_SearchElementPosition(ElementName := mpESQ^.Position);

// Check if ElementNumber is valid
IF meElementNumber > E_ElementNumber.E_BEGIN_ELEMENT AND 
   meElementNumber < E_ElementNumber.E_END_ELEMENT THEN			
	
	// Forward to element
	M_ProcessESQ := M_ProcessToElement(
						meElementNumber	:= meElementNumber, 
						meChannelSrc	:= meChannelSrc, 
						mMsgType		:= E_ITC_MsgTypeConv.ELEMENT_STATUS_REQUEST,
						mpData			:= mpESQ, 
						mLen			:= mLen);
						
// Check if ESQ was sent to a SubSystem
ELSIF F_EqualSisNames(Name1 := SubsystemRegistry.SubSystemName,
                      Name2 := mpESQ^.Position) THEN
									
	// Do for each ElementNumber
	FOR meElementNumber := E_ElementNumber.E_BEGIN_ELEMENT + 1 TO E_ElementNumber.E_END_Element - 1 DO
		// Forward
		M_ProcessToElement(
			meElementNumber	:= meElementNumber, 
			meChannelSrc	:= meChannelSrc, 
			mMsgType		:= E_ITC_MsgTypeConv.ELEMENT_STATUS_REQUEST,
			mpData			:= mpESQ, 
			mLen			:= mLen);
	END_FOR
ELSE
	ESR := ESR_Empty;
	// Unknown Position name received
	// ESR
	ESR.Position	:= mpESQ^.Position;
	ESR.ReturnCode	:= E_ErrorConv.ELEMENTNUMBER_UNKNOWN;

	// Reject telegram	
	M_SendData(
		meChannel := meChannelSrc,
		mMsgType  := E_ITC_MsgTypeConv.ELEMENT_STATUS_REPORT,
		mpData    := ADR(ESR),
		mLen	  := SIZEOF(ESR));
		
	// Unknown Position name received
	DebugMsg := CONCAT('ESQ - unknown Position name received: ', mpESQ^.Position);
	fbDebugMsg.M_SendErrorMsg(mMessage := DebugMsg);
END_IF
END_METHOD

METHOD PROTECTED M_ProcessFCQ : BOOL
(**************************************************************************************
 * 	Application		:	BoxControl Framework
 *	Revision		:	$Revision: 474929 $
 *	Revision date	:	$Date: 2021-04-08 12:45:11 +0200 (tor, 08 apr 2021) $
 *	Last changed by	:	$Author: b7gessa $
 *	URL				:	$URL: http://almscdc.swisslog.com/repo/SWPD/Development/BoxControlFramework/20_Release/tags/R1.12.0/01_Software/BCF/BCF/JumpStart/20_Product/10_BCF/11_Conv/11_Com/11_ITC/FB_ITC_Conveyor.TcPOU $
 *
 *	Purpose			:	Process a received Function Control Request.
 *
 * ------------------------------------------------------------------------------------
 *	Copyright Swisslog [IP AG], Switzerland. All rights reserved.
 * 
 * ------------------------------------------------------------------------------------
 *	
 * 	Revision History: 
 *
 * 	VERSION			DATE			INITIALS			DESCRIPTION
 *	0.1				01.01.2001		swl					Example
 *
 **************************************************************************************)
VAR_INPUT
	meChannelSrc		: E_MFCS_Channel; // Source communicaton channel
	mpFCQ				: POINTER TO ST_ITC_FCQ; // Pointer to FCQ
	mLen				: UDINT; // Data length
END_VAR

VAR
	mMsgPosition		: ST_PositionIdent; // Function position
	mrefObject			: REFERENCE TO FB_BaseObject; // Reference
END_VAR
// Initialize
M_ProcessFCQ := TRUE;

// Get position from message
mMsgPosition := F_SearchFunctionPosition(Position := mpFCQ^.Position);

// If a valid function was found with a valid zone
IF 	mMsgPosition.eFunctionNumber > E_FunctionNumber.F_BEGIN_FUNCTION AND 
	mMsgPosition.eFunctionNumber < E_FunctionNumber.F_END_FUNCTION AND 
	mMsgPosition.ZoneNumber >= 0 AND mMsgPosition.ZoneNumber <= NUMBER_OF_ZONES_PER_FUNCTION THEN
	
	// Forward to element
	M_ProcessFCQ := M_ProcessToFunction(
						meFunctionNumber	:= mMsgPosition.eFunctionNumber, 
						meChannelSrc		:= meChannelSrc, 
						mMsgType			:= E_ITC_MsgTypeConv.FUNCTION_CONTROL_REQUEST,
						mpData				:= mpFCQ, 
						mLen				:= mLen);
						
ELSE
	// FCR
	FCR.Position	:= mpFCQ^.Position;
	FCR.Code		:= mpFCQ^.Code;
	FCR.Variable	:= mpFCQ^.Variable;
	FCR.ReturnCode	:= E_ErrorConv.FUNCTIONNUMBER_UNKNOWN;

	// Reject telegram	
	M_SendData(
		meChannel := meChannelSrc,
		mMsgType  := E_ITC_MsgTypeConv.FUNCTION_CONTROL_REPLY,
		mpData    := ADR(FCR),
        mLen	  := SIZEOF(FCR));
		
	// Unknown Position name received 
	DebugMsg := CONCAT('FCQ, Unknown Position received: ', mpFCQ^.Position);
	fbDebugMsg.M_SendErrorMsg(mMessage := DebugMsg); 
END_IF
END_METHOD

METHOD PROTECTED M_ProcessFSQ : BOOL
(**************************************************************************************
 * 	Application		:	BoxControl Framework
 *	Revision		:	$Revision: 474929 $
 *	Revision date	:	$Date: 2021-04-08 12:45:11 +0200 (tor, 08 apr 2021) $
 *	Last changed by	:	$Author: b7gessa $
 *	URL				:	$URL: http://almscdc.swisslog.com/repo/SWPD/Development/BoxControlFramework/20_Release/tags/R1.12.0/01_Software/BCF/BCF/JumpStart/20_Product/10_BCF/11_Conv/11_Com/11_ITC/FB_ITC_Conveyor.TcPOU $
 *
 *	Purpose			:	Process a received position Status Request telegram.
 *
 * ------------------------------------------------------------------------------------
 *	Copyright Swisslog [IP AG], Switzerland. All rights reserved.
 * 
 * ------------------------------------------------------------------------------------
 *	
 * 	Revision History: 
 *
 * 	VERSION			DATE			INITIALS			DESCRIPTION
 *	0.1				01.01.2001		swl					Example
 *
 **************************************************************************************)
VAR_INPUT
	meChannelSrc		: E_MFCS_Channel; // Source communicaton channel
	mpFSQ				: POINTER TO ST_ITC_FSQ; // Pointer to FSQ
	mLen				: UDINT; // Data length
END_VAR

VAR
	mMsgPosition		: ST_PositionIdent; // Function position
	mrefObject			: REFERENCE TO FB_BaseObject; // Reference
END_VAR
// Initialize
M_ProcessFSQ := TRUE;

// Get position from message
mMsgPosition := F_SearchFunctionPosition(Position := mpFSQ^.Position);

// If a valid function was found with a valid zone
IF 	mMsgPosition.eFunctionNumber > E_FunctionNumber.F_BEGIN_FUNCTION AND 
	mMsgPosition.eFunctionNumber < E_FunctionNumber.F_END_FUNCTION AND 
	mMsgPosition.ZoneNumber >= 0 AND mMsgPosition.ZoneNumber <= NUMBER_OF_ZONES_PER_FUNCTION THEN

	// Forward to element
	M_ProcessFSQ := M_ProcessToFunction(
						meFunctionNumber	:= mMsgPosition.eFunctionNumber, 
						meChannelSrc		:= meChannelSrc, 
						mMsgType			:= E_ITC_MsgTypeConv.FUNCTION_STATUS_REQUEST,
						mpData				:= mpFSQ,
						mLen				:= mLen);

ELSE
	
	FSR := FSR_Empty;
	
	// FSR
	FSR.Position	:= mpFSQ^.Position;
	FSR.eReturnCode	:= E_ErrorConv.FUNCTIONNUMBER_UNKNOWN;

	// Reject telegram	
	M_SendData(
		meChannel := meChannelSrc,
		mMsgType  := E_ITC_MsgTypeConv.FUNCTION_STATUS_REPORT,
		mpData    := ADR(FSR),
		mLen	  := SIZEOF(FSR));
		
	// Unknown Position name received 
	DebugMsg := CONCAT('FSQ, Unknown Position received: ', mpFSQ^.Position);
	fbDebugMsg.M_SendErrorMsg(mMessage := DebugMsg); 
END_IF
END_METHOD

METHOD PROTECTED M_ProcessGCQ : BOOL
(**************************************************************************************
 * 	Application		:	BoxControl Framework
 *	Revision		:	$Revision: 474929 $
 *	Revision date	:	$Date: 2021-04-08 12:45:11 +0200 (tor, 08 apr 2021) $
 *	Last changed by	:	$Author: b7gessa $
 *	URL				:	$URL: http://almscdc.swisslog.com/repo/SWPD/Development/BoxControlFramework/20_Release/tags/R1.12.0/01_Software/BCF/BCF/JumpStart/20_Product/10_BCF/11_Conv/11_Com/11_ITC/FB_ITC_Conveyor.TcPOU $
 *
 *	Purpose			:	Process a received Group Control Request telegram.
 *
 * ------------------------------------------------------------------------------------
 *	Copyright Swisslog [IP AG], Switzerland. All rights reserved.
 * 
 * ------------------------------------------------------------------------------------
 *	
 * 	Revision History: 
 *
 * 	VERSION			DATE			INITIALS			DESCRIPTION
 *	0.1				01.01.2001		swl					Example
 *
 **************************************************************************************)
VAR_INPUT
	meChannelSrc		: E_MFCS_Channel; // Source communicaton channel
	mpGCQ				: POINTER TO ST_ITC_GCQ; // Pointer to GCQ
	mLen				: UDINT; // Data length
END_VAR

VAR
	meGroupNumber		: E_GroupNumber; // group number
END_VAR
// Initialize 
M_ProcessGCQ := TRUE;

// Find GropuNumber of telegram
meGroupNumber := F_SearchGroupNumber(GroupName := mpGCQ^.Position);
			
// Group number valid
IF meGroupNumber > E_GroupNumber.G_BEGIN_GROUP AND 
   meGroupNumber < E_GroupNumber.G_END_GROUP THEN	
				
	// Forward to group
	M_ProcessGCQ := M_ProcessToGroup(
						meGroupNumber	:= meGroupNumber, 
						meChannelSrc	:= meChannelSrc, 
						mMsgType		:= E_ITC_MsgTypeConv.GROUP_CONTROL_REQUEST,
						mpData			:= mpGCQ, 
						mLen			:= mLen);
				
// Check if GCQ was sent to a SubSystem
ELSIF F_EqualSisNames(Name1 := SubsystemRegistry.SubSystemName,
                      Name2 := mpGCQ^.Position) THEN
			
	// Do for each GroupNumber
	FOR meGroupNumber := E_GroupNumber.G_BEGIN_GROUP + 1 TO E_GroupNumber.G_END_GROUP - 1 DO
		// Check if group is a switching group
		IF GroupRegistry[meGroupNumber].eGroupType = E_GroupType.SG THEN
			M_ProcessToGroup(
				meGroupNumber	:= meGroupNumber, 
				meChannelSrc	:= meChannelSrc, 
				mMsgType		:= E_ITC_MsgTypeConv.GROUP_CONTROL_REQUEST,
				mpData			:= mpGCQ, 
				mLen 			:= mLen);
		END_IF
	END_FOR
ELSE
	
	// GCR
	GCR.GroupName	:= mpGCQ^.Position;
	GCR.Code		:= mpGCQ^.Code;
	GCR.Variable	:= mpGCQ^.Variable;
	GCR.ReturnCode	:= E_ErrorConv.GROUPNUMBER_UNKNOWN;

	// Reject telegram	
	M_SendData(
		meChannel := meChannelSrc,
		mMsgType  := E_ITC_MsgTypeConv.GROUP_CONTROL_REPLY,
		mpData    := ADR(GCR),
		mLen	  := SIZEOF(GCR));

	// Unknown Group name received
	DebugMsg := CONCAT('GCQ, unknown Group name received: ', mpGCQ^.Position);
	fbDebugMsg.M_SendErrorMsg(mMessage := DebugMsg);
END_IF
END_METHOD

METHOD PROTECTED M_ProcessGDQ : BOOL
(**************************************************************************************
 * 	Application		:	BoxControl Framework
 *	Revision		:	$Revision: 474929 $
 *	Revision date	:	$Date: 2021-04-08 12:45:11 +0200 (tor, 08 apr 2021) $
 *	Last changed by	:	$Author: b7gessa $
 *	URL				:	$URL: http://almscdc.swisslog.com/repo/SWPD/Development/BoxControlFramework/20_Release/tags/R1.12.0/01_Software/BCF/BCF/JumpStart/20_Product/10_BCF/11_Conv/11_Com/11_ITC/FB_ITC_Conveyor.TcPOU $
 *
 *	Purpose			:	Process a received Gathered Data Request telegram.
 *
 * ------------------------------------------------------------------------------------
 *	Copyright Swisslog [IP AG], Switzerland. All rights reserved.
 * 
 * ------------------------------------------------------------------------------------
 *	
 * 	Revision History: 
 *
 * 	VERSION			DATE			INITIALS			DESCRIPTION
 *	0.1				01.01.2001		swl					Example
 *
 **************************************************************************************)
VAR_INPUT
	meChannelSrc		: E_MFCS_Channel; // Source communicaton channel
	mpGDQ				: POINTER TO ST_ITC_GDQ; // Pointer to GDQ
	mLen				: UDINT; // Data length
END_VAR
VAR
	meFunctionPosition				: ST_PositionIdent; // Position
	meGroupNumber					: E_GroupNumber; // Group
	meElementNumber					: E_ElementNumber;//Element Number
	meSubsystem						: BOOL;	
	mReturnCode						: E_ErrorConv; // Error code
END_VAR
// Initialize
M_ProcessGDQ:= TRUE;

//Search Position
meFunctionPosition := F_SearchFunctionPosition(Position := mpGDQ^.Position);
meElementNumber    := F_SearchElementPosition(ElementName := mpGDQ^.Position);
meGroupNumber      := F_SearchGroupNumber(GroupName := mpGDQ^.Position);
meSubsystem 	   := F_EqualSisNames(Name1 := SubsystemRegistry.SubSystemName,
														        Name2 := mpGDQ^.Position);

// Check if Function is Target for Telgram 
IF meFunctionPosition.eFunctionNumber >F_BEGIN_FUNCTION AND
	meFunctionPosition.eFunctionNumber <F_END_FUNCTION THEN 
    // Forward to Function
	M_ProcessGDQ := M_ProcessToFunction(
						meFunctionNumber:= 	meFunctionPosition.eFunctionNumber, // Position
						meChannelSrc	:= meChannelSrc, 
						mpData			:= mpGDQ, 
						mMsgType		:= E_ITC_MsgTypeConv.GATHERED_DATA_REQUEST,
						mLen			:= mLen);
// Check if Element is Target for Telgram 
ELSIF meElementNumber > E_ElementNumber.E_BEGIN_ELEMENT AND 
      meElementNumber < E_ElementNumber.E_END_ELEMENT AND
      meFunctionPosition.eFunctionNumber = F_BEGIN_FUNCTION AND
      meFunctionPosition.ZoneNumber = 0 THEN 
	// Forward to element
	M_ProcessGDQ := M_ProcessToElement(
						meElementNumber	:= meElementNumber, 
						meChannelSrc	:= meChannelSrc, 
						mpData			:= mpGDQ, 
						mMsgType		:= E_ITC_MsgTypeConv.GATHERED_DATA_REQUEST,
						mLen			:= mLen);

// Check if Group is Target for Telgram 				
ELSIF  	meGroupNumber > E_GroupNumber.G_BEGIN_GROUP AND 
   		meGroupNumber < E_GroupNumber.G_END_GROUP   AND
		meElementNumber 					= E_BEGIN_ELEMENT AND 
      	meFunctionPosition.eFunctionNumber 	= F_BEGIN_FUNCTION AND
      	meFunctionPosition.ZoneNumber 		= 0 THEN 	   
			
		// Forward to Group
		M_ProcessGDQ := M_ProcessToGroup(
											meGroupNumber	:= meGroupNumber, // Groupnumber
											meChannelSrc	:= meChannelSrc, 
											mpData			:= mpGDQ, 
											mMsgType		:= E_ITC_MsgTypeConv.GATHERED_DATA_REQUEST,
											mLen			:= mLen);
	 
		
// Check if Subystem Target for Telgram 
ELSIF  meSubsystem AND
	   meGroupNumber = G_BEGIN_GROUP AND
	   meElementNumber = E_BEGIN_ELEMENT AND 
	   meFunctionPosition.eFunctionNumber = F_BEGIN_FUNCTION AND
	   meFunctionPosition.ZoneNumber = 0 THEN 	   	
		// Forward to Subsytem			
		M_ProcessGDQ := M_ProcessToSubsystem(
							meChannelSrc	:= meChannelSrc, 
							mpData			:= mpGDQ, 
							mMsgType		:= E_ITC_MsgTypeConv.GATHERED_DATA_REQUEST,
							mLen			:= mLen);
						
		
					
ELSE
	//Unknown position send DAR with Error Report	
	GDR := GDR_Empty;
	
	// DAR
	GDR.Position	:= mpGDQ^.Position;
	GDR.eReturnCode	:= E_ErrorConv.CONFIGURATION_ERROR;

	// Reject telegram	
	M_SendData(
		meChannel := meChannelSrc,
		mMsgType  := E_ITC_MsgTypeConv.GATHERED_DATA_REQUEST,
		mpData    := ADR(GDR),
		mLen	  := mLen );
		
	// Unknown Position name received
	DebugMsg := CONCAT('GDQ - unknown Position name received: ', mpGDQ^.Position);
	fbDebugMsg.M_SendErrorMsg(mMessage := DebugMsg);
END_IF
END_METHOD

METHOD PROTECTED M_ProcessGSQ : BOOL
(**************************************************************************************
 * 	Application		:	BoxControl Framework
 *	Revision		:	$Revision: 474929 $
 *	Revision date	:	$Date: 2021-04-08 12:45:11 +0200 (tor, 08 apr 2021) $
 *	Last changed by	:	$Author: b7gessa $
 *	URL				:	$URL: http://almscdc.swisslog.com/repo/SWPD/Development/BoxControlFramework/20_Release/tags/R1.12.0/01_Software/BCF/BCF/JumpStart/20_Product/10_BCF/11_Conv/11_Com/11_ITC/FB_ITC_Conveyor.TcPOU $
 *
 *	Purpose			:	Process a received Group Status Request telegram.
 *
 * ------------------------------------------------------------------------------------
 *	Copyright Swisslog [IP AG], Switzerland. All rights reserved.
 * 
 * ------------------------------------------------------------------------------------
 *	
 * 	Revision History: 
 *
 * 	VERSION			DATE			INITIALS			DESCRIPTION
 *	0.1				01.01.2001		swl					Example
 *
 **************************************************************************************)
VAR_INPUT
	meChannelSrc		: E_MFCS_Channel; // Source communicaton channel
	mpGSQ				: POINTER TO ST_ITC_GSQ; // Pointer to GSQ
	mLen				: UDINT; // Data length
END_VAR

VAR
	meGroupNumber		: E_GroupNumber; // group number
END_VAR
// Initialize
M_ProcessGSQ := TRUE;

// Find GropuNumber of telegram
meGroupNumber := F_SearchGroupNumber(GroupName := mpGSQ^.Position);
			
// Request was for a group
// Group number valid
IF meGroupNumber > E_GroupNumber.G_BEGIN_GROUP AND 
   meGroupNumber < E_GroupNumber.G_END_GROUP THEN	
						
	// Forward to group
	M_ProcessGSQ := M_ProcessToGroup(
						meGroupNumber	:= meGroupNumber, 
						meChannelSrc	:= meChannelSrc, 
						mMsgType		:= E_ITC_MsgTypeConv.GROUP_STATUS_REQUEST,
						mpData			:= mpGSQ,
						mLen			:= mLen);
					
// Check if GCQ was sent to a SubSystem
ELSIF F_EqualSisNames(Name1 := SubsystemRegistry.SubSystemName,
                      Name2 := mpGSQ^.Position) THEN
			
	// Do for each GroupNumber
	FOR meGroupNumber := E_GroupNumber.G_BEGIN_GROUP + 1 TO E_GroupNumber.G_END_GROUP - 1 DO
		
		M_ProcessToGroup(
			meGroupNumber	:= meGroupNumber, 
			meChannelSrc	:= meChannelSrc, 
			mMsgType		:= E_ITC_MsgTypeConv.GROUP_STATUS_REQUEST,
			mpData			:= mpGSQ, 
			mLen			:= mLen);
	END_FOR
	
ELSE
	GSR := GSR_Empty;
	
	// GSR
	GSR.GroupName	:= mpGSQ^.Position;
	GSR.eReturnCode	:= E_ErrorConv.GROUPNUMBER_UNKNOWN;

	// Reject telegram	
	M_SendData(
		meChannel := meChannelSrc,
		mMsgType  := E_ITC_MsgTypeConv.GROUP_STATUS_REPORT,
		mpData    := ADR(GSR),
		mLen	  := SIZEOF(GSR));
		
	// Unknown Group name received
	DebugMsg := CONCAT('GSQ, unknown Group name received: ', mpGSQ^.Position);
	fbDebugMsg.M_SendErrorMsg(mMessage := DebugMsg);
END_IF
END_METHOD

METHOD PROTECTED M_ProcessGVQ : BOOL
(**************************************************************************************
 * 	Application		:	BoxControl Framework
 *	Revision		:	$Revision: 474929 $
 *	Revision date	:	$Date: 2021-04-08 12:45:11 +0200 (tor, 08 apr 2021) $
 *	Last changed by	:	$Author: b7gessa $
 *	URL				:	$URL: http://almscdc.swisslog.com/repo/SWPD/Development/BoxControlFramework/20_Release/tags/R1.12.0/01_Software/BCF/BCF/JumpStart/20_Product/10_BCF/11_Conv/11_Com/11_ITC/FB_ITC_Conveyor.TcPOU $
 *
 *	Purpose			:	Process a received Global Variable Request telegram.
 *
 * ------------------------------------------------------------------------------------
 *	Copyright Swisslog [IP AG], Switzerland. All rights reserved.
 * 
 * ------------------------------------------------------------------------------------
 *	
 * 	Revision History: 
 *
 * 	VERSION			DATE			INITIALS			DESCRIPTION
 *	0.1				01.01.2001		swl					Example
 *
 **************************************************************************************)
VAR_INPUT
	meChannelSrc		: E_MFCS_Channel; // Source communicaton channel
	mpGVQ				: POINTER TO ST_ITC_GVQ; // Pointer to GVQ
	mLen				: UDINT; // Data length
END_VAR

VAR
	mIdx				: INT; // Iterator
	mError				: BOOL; // Error during processing
	mVar				: ARRAY[0..9] OF DINT; // Temporary variables
END_VAR
// Initialize
M_ProcessGVQ := TRUE;

// Initialize
mError := FALSE;

// Check borders
IF mpGVQ^.Number > GVR_Table.NUMBER_OF_GVR_SIGNALS OR
   mpGVQ^.Number < 1  OR
   mpGVQ^.Quantity < 1 OR
   mpGVQ^.Quantity > 10 THEN
	// Set error
	mError := TRUE;
END_IF

// If no error is active
IF NOT mError THEN
	// If perform action is selected
	IF mpGVQ^.Code = 1 OR mpGVQ^.Code = 2 THEN
		// Map values
		mVar[0] := mpGVQ^.Variable[0];
		mVar[1] := mpGVQ^.Variable[1];
		mVar[2] := mpGVQ^.Variable[2];
		mVar[3] := mpGVQ^.Variable[3];
		mVar[4] := mpGVQ^.Variable[4];
		mVar[5] := mpGVQ^.Variable[5];
		mVar[6] := mpGVQ^.Variable[6];
		mVar[7] := mpGVQ^.Variable[7];
		mVar[8] := mpGVQ^.Variable[8];
		mVar[9] := mpGVQ^.Variable[9];
	   
		// Go trough quantity
		FOR mIdx := 0 TO mpGVQ^.Quantity - 1 DO
			// Set values
			GlobalVariable[mpGVQ^.Number, mIdx] := mVar[mIdx];
		END_FOR
	END_IF
	
	// If report state is selected
	IF mpGVQ^.Code = 0 OR mpGVQ^.Code = 2 THEN
		GVR.Number := mpGVQ^.Number;
		GVR.Quantity := mpGVQ^.Quantity;
		
		// Go trough quantity
		FOR mIdx := 0 TO 9 DO
			// Set values
			GVR.Variable[mIdx] := 0;
		END_FOR
		
		FOR mIdx := 0 TO mpGVQ^.Quantity - 1 DO
			// Set values
			GVR.Variable[mIdx] := GlobalVariable[mpGVQ^.Number, mIdx];
		END_FOR

		GVR.ReturnCode := E_ErrorConv.NO_ERROR_CODE;
	
		M_SendData(
			meChannel := meChannelSrc, 
			mMsgType  := E_ITC_MsgTypeConv.GLOBAL_VARIABLE_REPORT, 
			mpData    := ADR(GVR),
			mLen	  := SIZEOF(GVR));
	END_IF
ELSE
	GVR.Number := mpGVQ^.Number;
	GVR.Quantity := mpGVQ^.Quantity;
	GVR.Variable[0] :=0;
	GVR.Variable[1] := 0;
	GVR.Variable[2] := 0;
	GVR.Variable[3] := 0;
	GVR.Variable[4] := 0;
	GVR.Variable[5] := 0;
	GVR.Variable[6] := 0;
	GVR.Variable[7] := 0;
	GVR.Variable[8] := 0;
	GVR.Variable[9] := 0;
	GVR.ReturnCode := E_ErrorConv.WRONG_VALUE;

	M_SendData(
		meChannel := meChannelSrc, 
		mMsgType  := E_ITC_MsgTypeConv.GLOBAL_VARIABLE_REPORT, 
		mpData    := ADR(GVR),
		mLen	  := SIZEOF(GVR));
END_IF
END_METHOD

METHOD PROTECTED M_ProcessIRQ : BOOL
(**************************************************************************************
 * 	Application		:	BoxControl Framework
 *	Revision		:	$Revision: 474929 $
 *	Revision date	:	$Date: 2021-04-08 12:45:11 +0200 (tor, 08 apr 2021) $
 *	Last changed by	:	$Author: b7gessa $
 *	URL				:	$URL: http://almscdc.swisslog.com/repo/SWPD/Development/BoxControlFramework/20_Release/tags/R1.12.0/01_Software/BCF/BCF/JumpStart/20_Product/10_BCF/11_Conv/11_Com/11_ITC/FB_ITC_Conveyor.TcPOU $
 *
 *	Purpose			:	Process a received I/O Status Request telegram.
 *
 * ------------------------------------------------------------------------------------
 *	Copyright Swisslog [IP AG], Switzerland. All rights reserved.
 * 
 * ------------------------------------------------------------------------------------
 *	
 * 	Revision History: 
 *
 * 	VERSION			DATE			INITIALS			DESCRIPTION
 *	0.1				01.01.2001		swl					Example
 *
 **************************************************************************************)
VAR_INPUT
	meChannelSrc		: E_MFCS_Channel; // Source communicaton channel
	mpIRQ				: POINTER TO ST_ITC_IRQ; // Pointer to IRQ
	mLen				: UDINT; // Data length
END_VAR


VAR
	mInformation		: STRING(NUMBER_OF_ISR_DATA_LENGTH); // Internal information
	mSignalNumber		: INT; // SignalNumber
	mIdx				: INT; // Internal cunter
	mByte				: BYTE; // Internal Byte
END_VAR
// Initialize
M_ProcessIRQ := TRUE;

// Init String
mInformation := '';

// Get the signal data for each block of 4 requested
// an mDataLength of 01 actually means get 4 bits
FOR mIdx := 1 TO mpIRQ^.DataLength BY 1 DO
	
	// Calculate base signal number
	mSignalNumber  := (((mIdx - 1) * 4) + mpIRQ^.StartSignalNumber);
	// Init Byte
	mByte := 0;

	// Check if we will remain in range of the ISR Signal numbers
	IF (mSignalNumber + 4) <= NUMBER_OF_ISR_SIGNALS THEN
		// Get the signal state for this group of 4 and put them in the correct bits
		mByte.0 := ISR_SignalType[mpIRQ^.SignalType].SignalNumber[mSignalNumber];
		mByte.1 := ISR_SignalType[mpIRQ^.SignalType].SignalNumber[mSignalNumber + 1];
		mByte.2 := ISR_SignalType[mpIRQ^.SignalType].SignalNumber[mSignalNumber + 2];
		mByte.3 := ISR_SignalType[mpIRQ^.SignalType].SignalNumber[mSignalNumber + 3];
	END_IF

	// Convert the resultant tByte to a value between '0' and 'F'
	fbFormatString (sFormat := '%X', arg1 := F_BYTE(mByte));

	// Add the ASCII result for this block of 4 bits to the ISR.Information string
	mInformation := CONCAT(mInformation, fbFormatString.sOut);
END_FOR

(* Information string should always be 99 chars long
   therefore pad mInformation with trailing zeros. *)
FOR mIdx := LEN(mInformation) TO NUMBER_OF_ISR_DATA_LENGTH DO
	mInformation := CONCAT(mInformation, '0');
END_FOR

// Collect data
ISR.DataLength := mpIRQ^.DataLength;
ISR.Information := mInformation;
ISR.SignalType := mpIRQ^.SignalType;
ISR.StartSignalNumber := mpIRQ^.StartSignalNumber;
ISR.ReturnCode := E_ErrorConv.NO_ERROR_CODE;

M_SendData(
	meChannel := meChannelSrc, 
	mMsgType  := E_ITC_MsgTypeConv.I_O_STATUS_REPORT, 
	mpData    := ADR(ISR),
	mLen	  := SIZEOF(ISR));
END_METHOD

METHOD PROTECTED M_ProcessMCQ : BOOL
(**************************************************************************************
 * 	Application		:	BoxControl Framework
 *	Revision		:	$Revision: 474929 $
 *	Revision date	:	$Date: 2021-04-08 12:45:11 +0200 (tor, 08 apr 2021) $
 *	Last changed by	:	$Author: b7gessa $
 *	URL				:	$URL: http://almscdc.swisslog.com/repo/SWPD/Development/BoxControlFramework/20_Release/tags/R1.12.0/01_Software/BCF/BCF/JumpStart/20_Product/10_BCF/11_Conv/11_Com/11_ITC/FB_ITC_Conveyor.TcPOU $
 *
 *	Purpose			:	Process a received Manual Control Request telegram.
 *
 * ------------------------------------------------------------------------------------
 *	Copyright Swisslog [IP AG], Switzerland. All rights reserved.
 * 
 * ------------------------------------------------------------------------------------
 *	
 * 	Revision History: 
 *
 * 	VERSION			DATE			INITIALS			DESCRIPTION
 *	0.1				01.01.2001		swl					Example
 *
 **************************************************************************************)
VAR_INPUT
	meChannelSrc		: E_MFCS_Channel; // Source communicaton channel
	mpMCQ				: POINTER TO ST_ITC_MCQ; // Pointer to MCQ
	mLen				: UDINT; // Data length
END_VAR

VAR
	meElementNumber			: E_ElementNumber; // PositionNumber
	mFunction				: ST_PositionIdent; // Function
END_VAR

// Initialize
M_ProcessMCQ := TRUE;

// Get element number
meElementNumber := F_SearchElementPosition(ElementName := mpMCQ^.Position);

// Get function
mFunction := F_SearchFunctionPosition(Position := mpMCQ^.Position);

// Valid ElementNumber was found
IF meElementNumber > E_ElementNumber.E_BEGIN_ELEMENT AND meElementNumber < E_ElementNumber.E_END_ELEMENT THEN

	// Forward to element
	M_ProcessMCQ := M_ProcessToElement(
						meElementNumber	:= meElementNumber, 
						meChannelSrc	:= meChannelSrc, 
						mMsgType		:= E_ITC_MsgTypeConv.MANUAL_CONTROL_REQUEST,
						mpData			:= mpMCQ,
						mLen			:= mLen);		
		
// Valid FunctionNumber was found
ELSIF mFunction.eFunctionNumber > E_FunctionNumber.F_BEGIN_FUNCTION AND 
      mFunction.eFunctionNumber < E_FunctionNumber.F_END_FUNCTION THEN
	
	// Forward to function
	M_ProcessMCQ := M_ProcessToFunction(
						meFunctionNumber	:= mFunction.eFunctionNumber, 
						meChannelSrc		:= meChannelSrc, 
						mMsgType			:= E_ITC_MsgTypeConv.MANUAL_CONTROL_REQUEST,
						mpData				:= mpMCQ,
						mLen				:= mLen);
	
ELSE
	// Unknown name received
	MCR := MCR_Empty;	

	MCR.Position := mpMCQ^.Position;
	MCR.Mode := E_PositionMode.UNKNOWN_MODE;
	MCR.Code := mpMCQ^.Code;
	MCR.eReturnCode := E_ErrorConv.WRONG_VALUE;

	// Reject telegram	
	M_SendData(
		meChannel := meChannelSrc,
		mMsgType  := E_ITC_MsgTypeConv.MANUAL_CONTROL_REPORT,
		mpData    := ADR(MCR),
		mLen	  := SIZEOF(MCR));
		
	// Unknown name received
	DebugMsg := CONCAT('MCQ, unknown Position name received: ', mpMCQ^.Position);
	fbDebugMsg.M_SendErrorMsg(mMessage := DebugMsg);
END_IF
END_METHOD

METHOD PROTECTED M_ProcessRAA : BOOL
(**************************************************************************************
 * 	Application		:	BoxControl Framework
 *	Revision		:	$Revision: 474929 $
 *	Revision date	:	$Date: 2021-04-08 12:45:11 +0200 (tor, 08 apr 2021) $
 *	Last changed by	:	$Author: b7gessa $
 *	URL				:	$URL: http://almscdc.swisslog.com/repo/SWPD/Development/BoxControlFramework/20_Release/tags/R1.12.0/01_Software/BCF/BCF/JumpStart/20_Product/10_BCF/11_Conv/11_Com/11_ITC/FB_ITC_Conveyor.TcPOU $
 *
 *	Purpose			:	Process a received Transport Task Assignment telegram for a robot.
 *
 * ------------------------------------------------------------------------------------
 *	Copyright Swisslog [IP AG], Switzerland. All rights reserved.
 * 
 * ------------------------------------------------------------------------------------
 *	
 * 	Revision History: 
 *
 * VERSION DATE         INITIALS     DESCRIPTION
 * 0.0     DD.MM.YYYY   (name)       (explain customized modifications)
 *
 **************************************************************************************)

//***********************************************************************************************************
VAR_INPUT
  meChannelSrc          : E_MFCS_Channel         := 0;     // Source communicaton channel
  mpRAA                 : POINTER TO ST_ITC_RAA  := 0;     // Pointer to RAA
  mLen                  : UDINT                  := 0;     // Data length
END_VAR

//***********************************************************************************************************
VAR
  eFunctionNumber       : E_FunctionNumber       := 0;
  eElementNumber        : E_ElementNumber        := 0;
  eGroupNumber          : E_GroupNumber          := 0;
  //-------------------------------------------------------------------------------------
  Subsystem             : BOOL                   := FALSE;
END_VAR

// parse and find requested position
eFunctionNumber:= F_FindFunction  (Name:= mpRAA^.Position);
eElementNumber := F_FindElement   (Name:= mpRAA^.Position);
eGroupNumber   := F_FindGroup     (Name:= mpRAA^.Position);
Subsystem      := F_CheckSubsystem(Name:= mpRAA^.Position);

// to function ?
IF eFunctionNumber <> E_FunctionNumber.F_BEGIN_FUNCTION THEN
	M_ProcessRAA:= M_ProcessToFunction(	meFunctionNumber:= eFunctionNumber, 
										meChannelSrc    := meChannelSrc, 
										mMsgType        := E_ITC_MsgTypeConv.ROBOT_ACTION_ASSIGNMENT,
										mpData          := mpRAA, 
										mLen            := mLen);
	// forwarding successful -> no debug message necessary here


// to element ?
ELSIF eElementNumber <> E_ElementNumber.E_BEGIN_ELEMENT THEN
	M_ProcessRAA:= M_ProcessToElement(	meElementNumber:= eElementNumber,
										meChannelSrc   := meChannelSrc, 
										mMsgType       := E_ITC_MsgTypeConv.ROBOT_ACTION_ASSIGNMENT,
										mpData         := mpRAA, 
										mLen           := mLen);
	// forwarding successful -> no debug message necessary here


// to group ?
ELSIF eGroupNumber <> E_GroupNumber.G_BEGIN_GROUP THEN
	M_ProcessRAA:= M_ProcessToGroup(meGroupNumber:= eGroupNumber,
									meChannelSrc := meChannelSrc, 
									mMsgType     := E_ITC_MsgTypeConv.ROBOT_ACTION_ASSIGNMENT,
									mpData       := mpRAA, 
									mLen         := mLen);
	// forwarding successful -> no debug message necessary here


// to subsystem ?
ELSIF Subsystem THEN
	M_ProcessRAA:= M_ProcessToSubsystem(meChannelSrc:= meChannelSrc, 
										mMsgType    := E_ITC_MsgTypeConv.ROBOT_ACTION_ASSIGNMENT,
										mpData      := mpRAA, 
										mLen        := mLen);
	// forwarding successful -> no debug message necessary here


//* unknown position -> fire error telegram
ELSE
  // reject telegram
	RAC.Position        := mpRAA^.Position;
	RAC.CommandDataIndex:= mpRAA^.CommandDataIndex;
	RAC.GroupID         := mpRAA^.GroupID;
	RAC.AssignmentID    := mpRAA^.AssignmentID;
	RAC.eReturnCode     := E_ErrorConv.FUNCTIONNUMBER_UNKNOWN;
	M_SendData(	meChannel:= meChannelSrc, 
				mMsgType := E_ITC_MsgTypeConv.ROBOT_ACTION_COMPLETE, 
				mpData   := ADR(RAC),
				mLen     := SIZEOF(RAC));	

	// debug message
	// example: '11-000-0000-00-0,  unknown position addressed,  telegram = RAA,  Position = 99-999-9999-99-9,  AssignmentID = 9999999'
	DebugMsg:= '';
	DebugMsg:= CONCAT(DebugMsg, F_AddDividerToSisString(SubsystemRegistry.SubsystemName));
	DebugMsg:= CONCAT(DebugMsg, ', unknown position addressed');
	DebugMsg:= CONCAT(DebugMsg, DebugTextBlocks.TELEGRAM);
	DebugMsg:= CONCAT(DebugMsg, 'RAA');
	DebugMsg:= CONCAT(DebugMsg, DebugTextBlocks.POSITION);
	DebugMsg:= CONCAT(DebugMsg, F_AddDividerToSisString(Name:= mpRAA^.Position)  );
	DebugMsg:= CONCAT(DebugMsg, DebugTextBlocks.ASSIGNMENTID);
	DebugMsg:= CONCAT(DebugMsg, UDINT_TO_STRING(mpRAA^.AssignmentID) );
	fbDebugMsg.M_SendErrorMsg(mMessage := DebugMsg);
	
	// forwarding to here ITC were possible so prevent error message from FB_SIS_MsgManager
	M_ProcessRAA:= TRUE;
END_IF
END_METHOD

METHOD PROTECTED M_ProcessRDQ : BOOL
(**************************************************************************************
 * 	Application		:	BoxControl Framework
 *	Revision		:	$Revision: 474929 $
 *	Revision date	:	$Date: 2021-04-08 12:45:11 +0200 (tor, 08 apr 2021) $
 *	Last changed by	:	$Author: b7gessa $
 *	URL				:	$URL: http://almscdc.swisslog.com/repo/SWPD/Development/BoxControlFramework/20_Release/tags/R1.12.0/01_Software/BCF/BCF/JumpStart/20_Product/10_BCF/11_Conv/11_Com/11_ITC/FB_ITC_Conveyor.TcPOU $
 *
 *	Purpose			:	Robot delete request
 *
 * ------------------------------------------------------------------------------------
 *	Copyright Swisslog [IP AG], Switzerland. All rights reserved.
 * 
 * ------------------------------------------------------------------------------------
 *	
 * 	Revision History: 
 *
 * 	VERSION			DATE			INITIALS			DESCRIPTION
 *	0.1				03.11.2015		Kay Röder			Example
 *
 **************************************************************************************)
VAR_INPUT
	meChannelSrc				: E_MFCS_Channel; // Source communicaton channel
	mpRDQ						: POINTER TO ST_ITC_RDQ; // Pointer to EDQ
	mLen						: UDINT; // Data length
END_VAR

VAR
	mMsgPosition		: ST_PositionIdent; // Function position
	mReturnCode 		: U_ErrorCode;
END_VAR
// Initialize
M_ProcessRDQ := TRUE;
	   
// Get position from message
mMsgPosition := F_SearchFunctionPosition(Position := mpRDQ^.Position);
	
// If a valid function was found with a valid zone
IF 	mMsgPosition.eFunctionNumber > E_FunctionNumber.F_BEGIN_FUNCTION AND 
	mMsgPosition.eFunctionNumber < E_FunctionNumber.F_END_FUNCTION AND 
	mMsgPosition.ZoneNumber >= 0 AND mMsgPosition.ZoneNumber <= NUMBER_OF_ZONES_PER_FUNCTION THEN
	
	// Forward to element
	M_ProcessRDQ := M_ProcessToFunction(
						meFunctionNumber	:= mMsgPosition.eFunctionNumber, 
						meChannelSrc		:= meChannelSrc, 
						mMsgType			:= E_ITC_MsgTypeConv.ROBOT_DELETE_REQUEST,
						mpData				:= mpRDQ, 
						mLen				:= mLen);
				
	DebugMsg := CONCAT('Robot Delete Assignment Request: ', UDINT_TO_STRING(mpRDQ^.AssignmentID));
	fbDebugMsg.M_SendInfoMsg(mMessage := DebugMsg);
 
ELSE
	mReturnCode.Conv := E_ErrorConv.FUNCTIONNUMBER_UNKNOWN; 
	
	// Reject telegram	
	RDR.Position := mpRDQ^.Position;
	RDR.CommandDataIndex := mpRDQ^.CommandDataIndex;
	RDR.GroupID := mpRDQ^.GroupID;
	RDR.AssignmentID := 0;
	RDR.ReturnCode := mReturnCode.Conv;

	M_SendData(
		meChannel := meChannelSrc, 
		mMsgType  := E_ITC_MsgTypeConv.ROBOT_DELETE_REPORT, 
		mpData    := ADR(RDR),
		mLen	  := SIZEOF(RDR));

	DebugMsg := CONCAT('Robot Delete Assignment Request: ', UDINT_TO_STRING(mpRDQ^.AssignmentID));
	DebugMsg := CONCAT(DebugMsg, 'has an invalid ITC config on RowPaQ-PLC-project');
	fbDebugMsg.M_SendErrorMsg(mMessage := DebugMsg);
END_IF
END_METHOD

METHOD PROTECTED M_ProcessSCQ : BOOL
(**************************************************************************************
 * 	Application		:	BoxControl Framework
 *	Revision		:	$Revision: 474929 $
 *	Revision date	:	$Date: 2021-04-08 12:45:11 +0200 (tor, 08 apr 2021) $
 *	Last changed by	:	$Author: b7gessa $
 *	URL				:	$URL: http://almscdc.swisslog.com/repo/SWPD/Development/BoxControlFramework/20_Release/tags/R1.12.0/01_Software/BCF/BCF/JumpStart/20_Product/10_BCF/11_Conv/11_Com/11_ITC/FB_ITC_Conveyor.TcPOU $
 *
 *	Purpose			:	Process a received Subsystem Control Request telegram.
 *
 * ------------------------------------------------------------------------------------
 *	Copyright Swisslog [IP AG], Switzerland. All rights reserved.
 * 
 * ------------------------------------------------------------------------------------
 *	
 * 	Revision History: 
 *
 * 	VERSION			DATE			INITIALS			DESCRIPTION
 *	0.1				01.01.2001		swl					Example
 *
 **************************************************************************************)
VAR_INPUT
	meChannelSrc		: E_MFCS_Channel; // Source communicaton channel
	mpSCQ				: POINTER TO ST_ITC_SCQ; // Pointer to SCQ
	mLen				: UDINT; // Data length
END_VAR
// Initialize 
M_ProcessSCQ := TRUE;

// Check if SubSystem is valid
IF F_EqualSisNames(Name1 := SubsystemRegistry.SubSystemName,
                   Name2 := mpSCQ^.SubsystemName) THEN
		
	// Forward to subsystem
	M_ProcessSCQ := M_ProcessToSubsystem(
						meChannelSrc	:= meChannelSrc, 
						mMsgType		:= E_ITC_MsgTypeConv.SUBSYSTEM_CONTROL_REQUEST,
						mpData			:= mpSCQ,
						mLen			:= mLen);		
ELSE
	// Unknown SubSystem number received
	SCR.SubsystemName	:= mpSCQ^.SubsystemName;
	SCR.Code			:= mpSCQ^.Code;
	SCR.Variable		:= mpSCQ^.Variable;
	SCR.ReturnCode		:= E_ErrorConv.SubsystemNUMBER_UNKNOWN;

	// Reject telegram	
	M_SendData(
		meChannel := meChannelSrc,
		mMsgType  := E_ITC_MsgTypeConv.SUBSYSTEM_CONTROL_REPLY,
		mpData    := ADR(SCR),
		mLen	  := SIZEOF(SCR));

	// Unknown SubSystem number received
	DebugMsg := CONCAT('SCQ, unknown SubSystem name received: ', mpSCQ^.SubsystemName);
	fbDebugMsg.M_SendErrorMsg(mMessage := DebugMsg);
END_IF
END_METHOD

METHOD PROTECTED M_ProcessSDO : BOOL
(**************************************************************************************
 * 	Application		:	BoxControl Framework
 *	Revision		:	$Revision: 474929 $
 *	Revision date	:	$Date: 2021-04-08 12:45:11 +0200 (tor, 08 apr 2021) $
 *	Last changed by	:	$Author: b7gessa $
 *	URL				:	$URL: http://almscdc.swisslog.com/repo/SWPD/Development/BoxControlFramework/20_Release/tags/R1.12.0/01_Software/BCF/BCF/JumpStart/20_Product/10_BCF/11_Conv/11_Com/11_ITC/FB_ITC_Conveyor.TcPOU $
 *
 *	Purpose			:	Process a received Set Digital Output telegram.
 *						Set or Reset the appropriate SDO signal number according 
 *						to the data in the telegram
 *
 * ------------------------------------------------------------------------------------
 *	Copyright Swisslog [IP AG], Switzerland. All rights reserved.
 * 
 * ------------------------------------------------------------------------------------
 *	
 * 	Revision History: 
 *
 * 	VERSION			DATE			INITIALS			DESCRIPTION
 *	0.1				01.01.2001		swl					Example
 *
 **************************************************************************************)
VAR_INPUT
	meChannelSrc		: E_MFCS_Channel; // Source communicaton channel
	mpSDO				: POINTER TO ST_ITC_SDO; // Pointer to SCQ
	mLen				: UDINT; // Data length
END_VAR
// Initialize
M_ProcessSDO := TRUE;

// Range check the SignalNumber
IF mpSDO^.SignalNumber > 0 THEN
	// Set SignalState
	SDOSignalNumber[mpSDO^.SignalNumber] := INT_TO_BOOL(mpSDO^.SignalState);
END_IF
END_METHOD

METHOD PROTECTED M_ProcessSIQ : BOOL
(**************************************************************************************
 * 	Application		:	BoxControl Framework
 *	Revision		:	$Revision: 474929 $
 *	Revision date	:	$Date: 2021-04-08 12:45:11 +0200 (tor, 08 apr 2021) $
 *	Last changed by	:	$Author: b7gessa $
 *	URL				:	$URL: http://almscdc.swisslog.com/repo/SWPD/Development/BoxControlFramework/20_Release/tags/R1.12.0/01_Software/BCF/BCF/JumpStart/20_Product/10_BCF/11_Conv/11_Com/11_ITC/FB_ITC_Conveyor.TcPOU $
 *
 *	Purpose			:	Process a received Scanner Information Request telegram.
 *
 * ------------------------------------------------------------------------------------
 *	Copyright Swisslog [IP AG], Switzerland. All rights reserved.
 * 
 * ------------------------------------------------------------------------------------
 *	
 * 	Revision History: 
 *
 * 	VERSION			DATE			INITIALS			DESCRIPTION
 *	0.1				01.01.2001		swl					Example
 *
 **************************************************************************************)
VAR_INPUT
	meChannelSrc		: E_MFCS_Channel; // Source communicaton channel
	mpSIQ				: POINTER TO ST_ITC_SIQ; // Pointer to SIQ
	mLen				: UDINT; // Data length
END_VAR

VAR
	mFunction			: ST_PositionIdent; // Function position
END_VAR
// Initialize
M_ProcessSIQ := TRUE;

//Find element function of telegram
mFunction := F_SearchFunctionPosition(Position := mpSIQ^.Position);

// If function number is valid
IF mFunction.eFunctionNumber > E_FunctionNumber.F_BEGIN_FUNCTION AND 
   mFunction.eFunctionNumber < E_FunctionNumber.F_END_FUNCTION THEN
   
	// Forward to function
	M_ProcessSIQ := M_ProcessToFunction(
						meFunctionNumber	:= mFunction.eFunctionNumber,
						meChannelSrc		:= meChannelSrc, 
						mMsgType			:= E_ITC_MsgTypeConv.SCANNER_INFORMATION_REQUEST,
						mpData				:= mpSIQ, 
						mLen				:= mLen);

ELSE
	// Unknown Position name received
	SIR.Position := mpSIQ^.Position;
	SIR.Code := mpSIQ^.Code;
	SIR.TU_ID := '';
	SIR.Counter1 := 0;
	SIR.Counter2 := 0;
	SIR.Counter3 := 0;
	SIR.Counter4 := 0;
	SIR.Counter5 := 0;
	SIR.eReturnCode := E_ErrorConv.FUNCTIONNUMBER_UNKNOWN;

	// Reject telegram	
	M_SendData(
		meChannel := meChannelSrc,
		mMsgType  := E_ITC_MsgTypeConv.SCANNER_INFORMATION_REPORT,
		mpData    := ADR(SIR),
		mLen	  := SIZEOF(SIR));

	// Unknown Position name received
	DebugMsg := CONCAT('SIQ, unknown Position name received: ', mpSIQ^.Position);
	fbDebugMsg.M_SendErrorMsg(mMessage := DebugMsg);	
END_IF
END_METHOD

METHOD PROTECTED M_ProcessSSQ : BOOL
(**************************************************************************************
 * 	Application		:	BoxControl Framework
 *	Revision		:	$Revision: 474929 $
 *	Revision date	:	$Date: 2021-04-08 12:45:11 +0200 (tor, 08 apr 2021) $
 *	Last changed by	:	$Author: b7gessa $
 *	URL				:	$URL: http://almscdc.swisslog.com/repo/SWPD/Development/BoxControlFramework/20_Release/tags/R1.12.0/01_Software/BCF/BCF/JumpStart/20_Product/10_BCF/11_Conv/11_Com/11_ITC/FB_ITC_Conveyor.TcPOU $
 *
 *	Purpose			:	Process a received Subsystem Status Request telegram.
 *
 * ------------------------------------------------------------------------------------
 *	Copyright Swisslog [IP AG], Switzerland. All rights reserved.
 * 
 * ------------------------------------------------------------------------------------
 *	
 * 	Revision History: 
 *
 * 	VERSION			DATE			INITIALS			DESCRIPTION
 *	0.1				01.01.2001		swl					Example
 *
 **************************************************************************************)
VAR_INPUT
	meChannelSrc		: E_MFCS_Channel; // Source communicaton channel
	mpSSQ				: POINTER TO ST_ITC_SSQ; // Pointer to SCQ
	mLen				: UDINT; // Data length
END_VAR
// Initialize
M_ProcessSSQ := TRUE;

// Check if SubSystem is valid
IF F_EqualSisNames(Name1 := SubsystemRegistry.SubsystemName,
                   Name2 := mpSSQ^.Position) THEN
		
		// Forward to subsystem
		M_ProcessSSQ := M_ProcessToSubsystem(
							meChannelSrc	:= meChannelSrc, 
							mMsgType		:= E_ITC_MsgTypeConv.SUBSYSTEM_STATUS_REQUEST,
							mpData			:= mpSSQ, 
							mLen			:= mLen);	
ELSE
	SSR := SSR_Empty;
	
